  STRUCT
   S711A_B_IDLE : STRUCT
    M_AUTO_SEL : BOOL ;
    M_MANUAL_SEL : BOOL ;
    M_READY_PB : BOOL ;
    M_AUTO_RUN_PB : BOOL ;
    M_WORK_COMP_SET_PB : BOOL ;
    M_WORK_COMP_RST_PB : BOOL ;
    M_HOME_POS_PB : BOOL ;
    M_TIP_DRESS_PB : BOOL ;
    LM_SLIDE_SEL : BOOL ;
    LM_SLIDE_LOCK_SEL : BOOL ;
    LM_PIN_SEL : BOOL ;
    LM_CLAMP1_SEL : BOOL ;
    LM_CLAMP2_SEL : BOOL ;
    LM_GUN1_ADV_RET_SEL : BOOL ;
    LM_GUN2_LATCH_SEL : BOOL ;
    LM_GUN2_ADV_RET_SEL : BOOL ;
    LM_GUN1_PRESS_SEL : BOOL ;
    LM_GUN2_PRESS_SEL : BOOL ;
    LM_GUN3_PRESS_SEL : BOOL ;
    LM_IDLE_LATCH_SEL : BOOL ;
    SPARE21 : BOOL ;
    SPARE22 : BOOL ;
    SPARE23 : BOOL ;
    SPARE24 : BOOL ;
    SPARE25 : BOOL ;
    SPARE26 : BOOL ;
    SPARE27 : BOOL ;
    SPARE28 : BOOL ;
    SPARE29 : BOOL ;
    SPARE30 : BOOL ;
    M_ADV_PB : BOOL ;
    M_RET_PB : BOOL ;
    TL_SLIDE_SEL : BOOL ;
    TL_SLIDE_LOCK_SEL : BOOL ;
    TL_PIN_SEL : BOOL ;
    TL_CLAMP_SEL : BOOL ;
    TL_GUN1_ADV_RET_SEL : BOOL ;
    TL_GUN2_ADV_RET_SEL : BOOL ;
    TL_GUN3_1_ADV_RET_SEL : BOOL ;
    TL_GUN3_2_ADV_RET_SEL : BOOL ;
    TL_GUN1_PRESS_SEL : BOOL ;
    TL_GUN2_PRESS_SEL : BOOL ;
    TL_GUN3_PRESS_SEL : BOOL ;
    TL_IDLE_LATCH_SEL : BOOL ;
    SPARE46 : BOOL ;
    SPARE47 : BOOL ;
    SPARE48 : BOOL ;
    SPARE49 : BOOL ;
    SPARE50 : BOOL ;
    SPARE51 : BOOL ;
    SPARE52 : BOOL ;
    SPARE53 : BOOL ;
    SPARE54 : BOOL ;
    SPARE55 : BOOL ;
    GUN_WELD_ON : BOOL ;
    GUN_TEST_ON : BOOL ;
    LM_SELECT : BOOL ;
    TL_SELECT : BOOL ;
    SPARE60 : BOOL ;
    SPARE61 : BOOL ;
    SPARE62 : BOOL ;
    SPARE63 : BOOL ;
    SPARE64 : BOOL ;
    SPARE65 : BOOL ;
    SPARE66 : BOOL ;
    SPARE67 : BOOL ;
    SPARE68 : BOOL ;
    SPARE69 : BOOL ;
    SPARE70 : BOOL ;
    SPARE71 : BOOL ;
    SPARE72 : BOOL ;
    SPARE73 : BOOL ;
    SPARE74 : BOOL ;
    SPARE75 : BOOL ;
    SPARE76 : BOOL ;
    SPARE77 : BOOL ;
    SPARE78 : BOOL ;
    SPARE79 : BOOL ;
    SPARE80 : BOOL ;
    SPARE81 : BOOL ;
    SPARE82 : BOOL ;
    SPARE83 : BOOL ;
    SPARE84 : BOOL ;
    SPARE85 : BOOL ;
    SPARE86 : BOOL ;
    SPARE87 : BOOL ;
    SPARE88 : BOOL ;
    SPARE89 : BOOL ;
    SPARE90 : BOOL ;
    SPARE91 : BOOL ;
    SPARE92 : BOOL ;
    SPARE93 : BOOL ;
    SPARE94 : BOOL ;
    SPARE95 : BOOL ;
    SPARE96 : BOOL ;
    SPARE97 : BOOL ;
    S711A_B_LM_AS_SEL : BOOL ;
    S711A_B_TL_AS_SEL : BOOL ;
    SPARE100 : BOOL ;
    SPARE101 : BOOL ;
    SPARE102 : BOOL ;
    SPARE103 : BOOL ;
    SPARE104 : BOOL ;
    SPARE105 : BOOL ;
    SPARE106 : BOOL ;
    SPARE107 : BOOL ;
    SPARE108 : BOOL ;
    SPARE109 : BOOL ;
    SPARE110 : BOOL ;
    SPARE111 : BOOL ;
    SPARE112 : BOOL ;
    SPARE113 : BOOL ;
    SPARE114 : BOOL ;
    SPARE115 : BOOL ;
    SPARE116 : BOOL ;
    SPARE117 : BOOL ;
    SPARE118 : BOOL ;
    SPARE119 : BOOL ;
    SPARE120 : BOOL ;
    SPARE121 : BOOL ;
    SPARE122 : BOOL ;
    SPARE123 : BOOL ;
    SPARE124 : BOOL ;
    SPARE125 : BOOL ;
    SPARE126 : BOOL ;
    SPARE127 : BOOL ;
    SPARE128 : BOOL ;
    SPARE129 : BOOL ;
    SPARE130 : BOOL ;
    SPARE131 : BOOL ;
    SPARE132 : BOOL ;
    SPARE133 : BOOL ;
    SPARE134 : BOOL ;
    SPARE135 : BOOL ;
    SPARE136 : BOOL ;
    SPARE137 : BOOL ;
    SPARE138 : BOOL ;
    SPARE139 : BOOL ;
    SPARE140 : BOOL ;
    SPARE141 : BOOL ;
    SPARE142 : BOOL ;
    SPARE143 : BOOL ;
    SPARE144 : BOOL ;
    SPARE145 : BOOL ;
    SPARE146 : BOOL ;
    SPARE147 : BOOL ;
    SPARE148 : BOOL ;
    SPARE149 : BOOL ;
    SPARE150 : BOOL ;
    SPARE151 : BOOL ;
    SPARE152 : BOOL ;
    SPARE153 : BOOL ;
    SPARE154 : BOOL ;
    SPARE155 : BOOL ;
    SPARE156 : BOOL ;
    SPARE157 : BOOL ;
    SPARE158 : BOOL ;
    SPARE159 : BOOL ;
    SPARE160 : BOOL ;
    SPARE161 : BOOL ;
    LM_SLIDE_ADV_LP : WORD ;
    LM_SLIDE_RET_LP : WORD ;
    LM_SLIDE_LOCK_ADV_LP : WORD ;
    LM_SLIDE_LOCK_RET_LP : WORD ;
    LM_PIN_UP_LP : WORD ;
    LM_PIN_DOWN_LP : WORD ;
    LM_CLAMP1_ADV_LP : WORD ;
    LM_CLAMP1_RET_LP : WORD ;
    LM_CLAMP2_ADV_LP : WORD ;
    LM_CLAMP2_RET_LP : WORD ;
    LM_GUN1_ADV_LP : WORD ;
    LM_GUN1_RET_LP : WORD ;
    LM_GUN2_LATCH_ADV_LP : WORD ;
    LM_GUN2_LATCH_RET_LP : WORD ;
    LM_GUN2_ADV_LP : WORD ;
    LM_GUN2_RET_LP : WORD ;
    LM_GUN1_PRESS_LP : WORD ;
    LM_GUN1_OPEN_LP : WORD ;
    LM_GUN2_PRESS_LP : WORD ;
    LM_GUN2_OPEN_LP : WORD ;
    LM_GUN3_PRESS_LP : WORD ;
    LM_GUN3_OPEN_LP : WORD ;
    LM_IDLE_LATCH_ADV_LP : WORD ;
    LM_IDLE_LATCH_RET_LP : WORD ;
    SP_WORD36 : WORD ;
    SP_WORD37 : WORD ;
    SP_WORD38 : WORD ;
    SP_WORD39 : WORD ;
    SP_WORD40 : WORD ;
    SP_WORD41 : WORD ;
    SP_WORD42 : WORD ;
    SP_WORD43 : WORD ;
    SP_WORD44 : WORD ;
    SP_WORD45 : WORD ;
    SP_WORD46 : WORD ;
    SP_WORD47 : WORD ;
    SP_WORD48 : WORD ;
    SP_WORD49 : WORD ;
    SP_WORD50 : WORD ;
    SP_WORD51 : WORD ;
    TL_SLIDE_ADV_LP : WORD ;
    TL_SLIDE_RET_LP : WORD ;
    TL_SLIDE_LOCK_ADV_LP : WORD ;
    TL_SLIDE_LOCK_RET_LP : WORD ;
    TL_PIN_UP_LP : WORD ;
    TL_PIN_DOWN_LP : WORD ;
    TL_CLAMP1_ADV_LP : WORD ;
    TL_CLAMP1_RET_LP : WORD ;
    TL_CLAMP2_ADV_LP : WORD ;
    TL_CLAMP2_RET_LP : WORD ;
    TL_GUN1_ADV_LP : WORD ;
    TL_GUN1_RET_LP : WORD ;
    TL_GUN2_ADV_LP : WORD ;
    TL_GUN2_RET_LP : WORD ;
    TL_GUN3_1_ADV_LP : WORD ;
    TL_GUN3_1_RET_LP : WORD ;
    TL_GUN3_2_ADV_LP : WORD ;
    TL_GUN3_2_RET_LP : WORD ;
    TL_GUN1_PRESS_LP : WORD ;
    TL_GUN1_OPEN_LP : WORD ;
    TL_GUN2_PRESS_LP : WORD ;
    TL_GUN2_OPEN_LP : WORD ;
    TL_GUN3_PRESS_LP : WORD ;
    TL_GUN3_OPEN_LP : WORD ;
    TL_IDLE_PIN_UP_LP : WORD ;
    TL_IDLE_PIN_DOWN_LP : WORD ;
    TL_IDLE_LATCH_ADV_LP : WORD ;
    TL_IDLE_LATCH_RET_LP : WORD ;
    SP_WORD80 : WORD ;
    SP_WORD81 : WORD ;
    SP_WORD82 : WORD ;
    SP_WORD83 : WORD ;
    SP_WORD84 : WORD ;
    SP_WORD85 : WORD ;
    SP_WORD86 : WORD ;
    SP_WORD87 : WORD ;
    SP_WORD88 : WORD ;
    SP_WORD89 : WORD ;
    SP_WORD90 : WORD ;
    SP_WORD91 : WORD ;
    SP_WORD92 : WORD ;
    SP_WORD93 : WORD ;
    SP_WORD94 : WORD ;
    SP_WORD95 : WORD ;
    SP_WORD96 : WORD ;
    SP_WORD97 : WORD ;
    SP_WORD98 : WORD ;
    SP_WORD99 : WORD ;
    SP_WORD100 : WORD ;
    SP_WORD101 : WORD ;
   END_STRUCT ;
   S711_COMPL : STRUCT
    M_AUTO_SEL : BOOL ;
    M_MANUAL_SEL : BOOL ;
    M_READY_PB : BOOL ;
    M_AUTO_RUN_PB : BOOL ;
    M_WORK_COMP_SET_PB : BOOL ;
    M_WORK_COMP_RST_PB : BOOL ;
    M_HOME_POS_PB : BOOL ;
    M_TIP_DRESS_PB : BOOL ;
    INDEX_LOCK_SEL : BOOL ;
    INDEX_TURN_RETURN_SEL : BOOL ;
    LM_BT_CHANGE_SEL : BOOL ;
    TL_BT_CHANGE_SEL : BOOL ;
    TL_PIN_SEL : BOOL ;
    LM_PIN_SEL : BOOL ;
    LM_CLAMP_SEL : BOOL ;
    INDEX_LM_CLAMP_SEL : BOOL ;
    SPARE17 : BOOL ;
    SPARE18 : BOOL ;
    SPARE19 : BOOL ;
    SPARE20 : BOOL ;
    SPARE21 : BOOL ;
    SPARE22 : BOOL ;
    SPARE23 : BOOL ;
    SPARE24 : BOOL ;
    SPARE25 : BOOL ;
    SPARE26 : BOOL ;
    SPARE27 : BOOL ;
    SPARE28 : BOOL ;
    SPARE29 : BOOL ;
    SPARE30 : BOOL ;
    M_ADV_PB : BOOL ;
    M_RET_PB : BOOL ;
    SPARE34 : BOOL ;
    SPARE35 : BOOL ;
    SPARE36 : BOOL ;
    SPARE37 : BOOL ;
    SPARE38 : BOOL ;
    SPARE39 : BOOL ;
    SPARE40 : BOOL ;
    SPARE41 : BOOL ;
    SPARE42 : BOOL ;
    SPARE43 : BOOL ;
    SPARE44 : BOOL ;
    SPARE45 : BOOL ;
    SPARE46 : BOOL ;
    SPARE47 : BOOL ;
    SPARE48 : BOOL ;
    SPARE49 : BOOL ;
    SPARE50 : BOOL ;
    SPARE51 : BOOL ;
    SPARE52 : BOOL ;
    SPARE53 : BOOL ;
    SPARE54 : BOOL ;
    SPARE55 : BOOL ;
    SPARE56 : BOOL ;
    SPARE57 : BOOL ;
    SPARE58 : BOOL ;
    SPARE59 : BOOL ;
    SPARE60 : BOOL ;
    SPARE61 : BOOL ;
    SPARE62 : BOOL ;
    SPARE63 : BOOL ;
    SPARE64 : BOOL ;
    SPARE65 : BOOL ;
    SPARE66 : BOOL ;
    SPARE67 : BOOL ;
    SPARE68 : BOOL ;
    SPARE69 : BOOL ;
    SPARE70 : BOOL ;
    SPARE71 : BOOL ;
    SPARE72 : BOOL ;
    SPARE73 : BOOL ;
    SPARE74 : BOOL ;
    SPARE75 : BOOL ;
    SPARE76 : BOOL ;
    SPARE77 : BOOL ;
    SPARE78 : BOOL ;
    SPARE79 : BOOL ;
    SPARE80 : BOOL ;
    SPARE81 : BOOL ;
    SPARE82 : BOOL ;
    SPARE83 : BOOL ;
    SPARE84 : BOOL ;
    SPARE85 : BOOL ;
    SPARE86 : BOOL ;
    SPARE87 : BOOL ;
    SPARE88 : BOOL ;
    SPARE89 : BOOL ;
    SPARE90 : BOOL ;
    SPARE91 : BOOL ;
    SPARE92 : BOOL ;
    SPARE93 : BOOL ;
    SPARE94 : BOOL ;
    SPARE95 : BOOL ;
    SPARE96 : BOOL ;
    SPARE97 : BOOL ;
    SPARE98 : BOOL ;
    SPARE99 : BOOL ;
    SPARE100 : BOOL ;
    SPARE101 : BOOL ;
    SPARE102 : BOOL ;
    SPARE103 : BOOL ;
    SPARE104 : BOOL ;
    SPARE105 : BOOL ;
    SPARE106 : BOOL ;
    SPARE107 : BOOL ;
    SPARE108 : BOOL ;
    SPARE109 : BOOL ;
    SPARE110 : BOOL ;
    SPARE111 : BOOL ;
    SPARE112 : BOOL ;
    SPARE113 : BOOL ;
    SPARE114 : BOOL ;
    SPARE115 : BOOL ;
    SPARE116 : BOOL ;
    SPARE117 : BOOL ;
    SPARE118 : BOOL ;
    SPARE119 : BOOL ;
    SPARE120 : BOOL ;
    SPARE121 : BOOL ;
    SPARE122 : BOOL ;
    SPARE123 : BOOL ;
    SPARE124 : BOOL ;
    SPARE125 : BOOL ;
    SPARE126 : BOOL ;
    SPARE127 : BOOL ;
    SPARE128 : BOOL ;
    SPARE129 : BOOL ;
    SPARE130 : BOOL ;
    SPARE131 : BOOL ;
    SPARE132 : BOOL ;
    SPARE133 : BOOL ;
    SPARE134 : BOOL ;
    SPARE135 : BOOL ;
    SPARE136 : BOOL ;
    SPARE137 : BOOL ;
    SPARE138 : BOOL ;
    SPARE139 : BOOL ;
    SPARE140 : BOOL ;
    SPARE141 : BOOL ;
    SPARE142 : BOOL ;
    SPARE143 : BOOL ;
    SPARE144 : BOOL ;
    SPARE145 : BOOL ;
    SPARE146 : BOOL ;
    SPARE147 : BOOL ;
    SPARE148 : BOOL ;
    SPARE149 : BOOL ;
    SPARE150 : BOOL ;
    SPARE151 : BOOL ;
    SPARE152 : BOOL ;
    SPARE153 : BOOL ;
    SPARE154 : BOOL ;
    SPARE155 : BOOL ;
    SPARE156 : BOOL ;
    SPARE157 : BOOL ;
    SPARE158 : BOOL ;
    SPARE159 : BOOL ;
    SPARE160 : BOOL ;
    SPARE161 : BOOL ;
    INDEX_LOCK_ADV_LP : WORD ;
    INDEX_LOCK_RET_LP : WORD ;
    INDEX_TURN_LP : WORD ;
    INDEX_RETURN_LP : WORD ;
    LM_BT_CHANGE_ADV_LP : WORD ;
    LM_BT_CHANGE_RET_LP : WORD ;
    TL_BT_CHANGE_ADV_LP : WORD ;
    TL_BT_CHANGE_RET_LP : WORD ;
    TL_PIN_UP_LP : WORD ;
    TL_PIN_DOWN_LP : WORD ;
    LM_PIN_UP_LP : WORD ;
    LM_PIN_DOWN_LP : WORD ;
    LM_CLAMP_ADV_LP : WORD ;
    LM_CLAMP_RET_LP : WORD ;
    INDEX_LM_CLAMP_ADV_LP : WORD ;
    INDEX_LM_CLAMP_RET_LP : WORD ;
    INDEX_LM_PIN_UP_LP : WORD ;
    INDEX_LM_PIN_DOWN_LP : WORD ;
    SP_WORD29 : WORD ;
    SP_WORD30 : WORD ;
    SP_WORD31 : WORD ;
    SP_WORD32 : WORD ;
    SP_WORD33 : WORD ;
    SP_WORD34 : WORD ;
    SP_WORD35 : WORD ;
    SP_WORD36 : WORD ;
    SP_WORD37 : WORD ;
    SP_WORD38 : WORD ;
    SP_WORD39 : WORD ;
    SP_WORD40 : WORD ;
    SP_WORD41 : WORD ;
    SP_WORD42 : WORD ;
    SP_WORD43 : WORD ;
    SP_WORD44 : WORD ;
    SP_WORD45 : WORD ;
    SP_WORD46 : WORD ;
    SP_WORD47 : WORD ;
    SP_WORD49 : WORD ;
    SP_WORD50 : WORD ;
    SP_WORD51 : WORD ;
    INR_PLT3_UP_LP : WORD ;
    INR_PLT3_DOWN_LP : WORD ;
    INR_PLT3_LOCK_ADV_LP : WORD ;
    INR_PLT3_LOCK_RET_LP : WORD ;
    INR_PLT4_UP_LP : WORD ;
    INR_PLT4_DOWN_LP : WORD ;
    INR_PLT4_LOCK_ADV_LP : WORD ;
    INR_PLT4_LOCK_RET_LP : WORD ;
    INR_PLT5_UP_LP : WORD ;
    INR_PLT5_DOWN_LP : WORD ;
    INR_PLT5_LOCK_ADV_LP : WORD ;
    INR_PLT5_LOCK_RET_LP : WORD ;
    SP_WORD64 : WORD ;
    SP_WORD65 : WORD ;
    SP_WORD66 : WORD ;
    SP_WORD67 : WORD ;
    SP_WORD68 : WORD ;
    SP_WORD69 : WORD ;
    SP_WORD70 : WORD ;
    SP_WORD71 : WORD ;
    SP_WORD72 : WORD ;
    SP_WORD73 : WORD ;
    SP_WORD74 : WORD ;
    SP_WORD75 : WORD ;
    SP_WORD76 : WORD ;
    SP_WORD77 : WORD ;
    SP_WORD78 : WORD ;
    SP_WORD79 : WORD ;
    SP_WORD80 : WORD ;
    SP_WORD81 : WORD ;
    SP_WORD82 : WORD ;
    SP_WORD83 : WORD ;
    SP_WORD84 : WORD ;
    SP_WORD85 : WORD ;
    SP_WORD86 : WORD ;
    SP_WORD87 : WORD ;
    SP_WORD88 : WORD ;
    SP_WORD89 : WORD ;
    SP_WORD90 : WORD ;
    SP_WORD91 : WORD ;
    SP_WORD92 : WORD ;
    SP_WORD93 : WORD ;
    SP_WORD94 : WORD ;
    SP_WORD95 : WORD ;
    SP_WORD96 : WORD ;
    SP_WORD97 : WORD ;
    SP_WORD98 : WORD ;
    SP_WORD99 : WORD ;
    SP_WORD100 : WORD ;
    SP_WORD101 : WORD ;
   END_STRUCT ;
  END_STRUCT ;
BEGIN
   S711A_B_IDLE.M_AUTO_SEL := FALSE;
   S711A_B_IDLE.M_MANUAL_SEL := FALSE;
   S711A_B_IDLE.M_READY_PB := FALSE;
   S711A_B_IDLE.M_AUTO_RUN_PB := FALSE;
   S711A_B_IDLE.M_WORK_COMP_SET_PB := FALSE;
   S711A_B_IDLE.M_WORK_COMP_RST_PB := FALSE;
   S711A_B_IDLE.M_HOME_POS_PB := FALSE;
   S711A_B_IDLE.M_TIP_DRESS_PB := FALSE;
   S711A_B_IDLE.LM_SLIDE_SEL := FALSE;
   S711A_B_IDLE.LM_SLIDE_LOCK_SEL := FALSE;
   S711A_B_IDLE.LM_PIN_SEL := FALSE;
   S711A_B_IDLE.LM_CLAMP1_SEL := FALSE;
   S711A_B_IDLE.LM_CLAMP2_SEL := FALSE;
   S711A_B_IDLE.LM_GUN1_ADV_RET_SEL := FALSE;
   S711A_B_IDLE.LM_GUN2_LATCH_SEL := FALSE;
   S711A_B_IDLE.LM_GUN2_ADV_RET_SEL := FALSE;
   S711A_B_IDLE.LM_GUN1_PRESS_SEL := FALSE;
   S711A_B_IDLE.LM_GUN2_PRESS_SEL := FALSE;
   S711A_B_IDLE.LM_GUN3_PRESS_SEL := FALSE;
   S711A_B_IDLE.LM_IDLE_LATCH_SEL := FALSE;
   S711A_B_IDLE.SPARE21 := FALSE;
   S711A_B_IDLE.SPARE22 := FALSE;
   S711A_B_IDLE.SPARE23 := FALSE;
   S711A_B_IDLE.SPARE24 := FALSE;
   S711A_B_IDLE.SPARE25 := FALSE;
   S711A_B_IDLE.SPARE26 := FALSE;
   S711A_B_IDLE.SPARE27 := FALSE;
   S711A_B_IDLE.SPARE28 := FALSE;
   S711A_B_IDLE.SPARE29 := FALSE;
   S711A_B_IDLE.SPARE30 := FALSE;
   S711A_B_IDLE.M_ADV_PB := FALSE;
   S711A_B_IDLE.M_RET_PB := FALSE;
   S711A_B_IDLE.TL_SLIDE_SEL := FALSE;
   S711A_B_IDLE.TL_SLIDE_LOCK_SEL := FALSE;
   S711A_B_IDLE.TL_PIN_SEL := FALSE;
   S711A_B_IDLE.TL_CLAMP_SEL := FALSE;
   S711A_B_IDLE.TL_GUN1_ADV_RET_SEL := FALSE;
   S711A_B_IDLE.TL_GUN2_ADV_RET_SEL := FALSE;
   S711A_B_IDLE.TL_GUN3_1_ADV_RET_SEL := FALSE;
   S711A_B_IDLE.TL_GUN3_2_ADV_RET_SEL := FALSE;
   S711A_B_IDLE.TL_GUN1_PRESS_SEL := FALSE;
   S711A_B_IDLE.TL_GUN2_PRESS_SEL := FALSE;
   S711A_B_IDLE.TL_GUN3_PRESS_SEL := FALSE;
   S711A_B_IDLE.TL_IDLE_LATCH_SEL := FALSE;
   S711A_B_IDLE.SPARE46 := FALSE;
   S711A_B_IDLE.SPARE47 := FALSE;
   S711A_B_IDLE.SPARE48 := FALSE;
   S711A_B_IDLE.SPARE49 := FALSE;
   S711A_B_IDLE.SPARE50 := FALSE;
   S711A_B_IDLE.SPARE51 := FALSE;
   S711A_B_IDLE.SPARE52 := FALSE;
   S711A_B_IDLE.SPARE53 := FALSE;
   S711A_B_IDLE.SPARE54 := FALSE;
   S711A_B_IDLE.SPARE55 := FALSE;
   S711A_B_IDLE.GUN_WELD_ON := FALSE;
   S711A_B_IDLE.GUN_TEST_ON := FALSE;
   S711A_B_IDLE.LM_SELECT := FALSE;
   S711A_B_IDLE.TL_SELECT := FALSE;
   S711A_B_IDLE.SPARE60 := FALSE;
   S711A_B_IDLE.SPARE61 := FALSE;
   S711A_B_IDLE.SPARE62 := FALSE;
   S711A_B_IDLE.SPARE63 := FALSE;
   S711A_B_IDLE.SPARE64 := FALSE;
   S711A_B_IDLE.SPARE65 := FALSE;
   S711A_B_IDLE.SPARE66 := FALSE;
   S711A_B_IDLE.SPARE67 := FALSE;
   S711A_B_IDLE.SPARE68 := FALSE;
   S711A_B_IDLE.SPARE69 := FALSE;
   S711A_B_IDLE.SPARE70 := FALSE;
   S711A_B_IDLE.SPARE71 := FALSE;
   S711A_B_IDLE.SPARE72 := FALSE;
   S711A_B_IDLE.SPARE73 := FALSE;
   S711A_B_IDLE.SPARE74 := FALSE;
   S711A_B_IDLE.SPARE75 := FALSE;
   S711A_B_IDLE.SPARE76 := FALSE;
   S711A_B_IDLE.SPARE77 := FALSE;
   S711A_B_IDLE.SPARE78 := FALSE;
   S711A_B_IDLE.SPARE79 := FALSE;
   S711A_B_IDLE.SPARE80 := FALSE;
   S711A_B_IDLE.SPARE81 := FALSE;
   S711A_B_IDLE.SPARE82 := FALSE;
   S711A_B_IDLE.SPARE83 := FALSE;
   S711A_B_IDLE.SPARE84 := FALSE;
   S711A_B_IDLE.SPARE85 := FALSE;
   S711A_B_IDLE.SPARE86 := FALSE;
   S711A_B_IDLE.SPARE87 := FALSE;
   S711A_B_IDLE.SPARE88 := FALSE;
   S711A_B_IDLE.SPARE89 := FALSE;
   S711A_B_IDLE.SPARE90 := FALSE;
   S711A_B_IDLE.SPARE91 := FALSE;
   S711A_B_IDLE.SPARE92 := FALSE;
   S711A_B_IDLE.SPARE93 := FALSE;
   S711A_B_IDLE.SPARE94 := FALSE;
   S711A_B_IDLE.SPARE95 := FALSE;
   S711A_B_IDLE.SPARE96 := FALSE;
   S711A_B_IDLE.SPARE97 := FALSE;
   S711A_B_IDLE.S711A_B_LM_AS_SEL := FALSE;
   S711A_B_IDLE.S711A_B_TL_AS_SEL := FALSE;
   S711A_B_IDLE.SPARE100 := FALSE;
   S711A_B_IDLE.SPARE101 := FALSE;
   S711A_B_IDLE.SPARE102 := FALSE;
   S711A_B_IDLE.SPARE103 := FALSE;
   S711A_B_IDLE.SPARE104 := FALSE;
   S711A_B_IDLE.SPARE105 := FALSE;
   S711A_B_IDLE.SPARE106 := FALSE;
   S711A_B_IDLE.SPARE107 := FALSE;
   S711A_B_IDLE.SPARE108 := FALSE;
   S711A_B_IDLE.SPARE109 := FALSE;
   S711A_B_IDLE.SPARE110 := FALSE;
   S711A_B_IDLE.SPARE111 := FALSE;
   S711A_B_IDLE.SPARE112 := FALSE;
   S711A_B_IDLE.SPARE113 := FALSE;
   S711A_B_IDLE.SPARE114 := FALSE;
   S711A_B_IDLE.SPARE115 := FALSE;
   S711A_B_IDLE.SPARE116 := FALSE;
   S711A_B_IDLE.SPARE117 := FALSE;
   S711A_B_IDLE.SPARE118 := FALSE;
   S711A_B_IDLE.SPARE119 := FALSE;
   S711A_B_IDLE.SPARE120 := FALSE;
   S711A_B_IDLE.SPARE121 := FALSE;
   S711A_B_IDLE.SPARE122 := FALSE;
   S711A_B_IDLE.SPARE123 := FALSE;
   S711A_B_IDLE.SPARE124 := FALSE;
   S711A_B_IDLE.SPARE125 := FALSE;
   S711A_B_IDLE.SPARE126 := FALSE;
   S711A_B_IDLE.SPARE127 := FALSE;
   S711A_B_IDLE.SPARE128 := FALSE;
   S711A_B_IDLE.SPARE129 := FALSE;
   S711A_B_IDLE.SPARE130 := FALSE;
   S711A_B_IDLE.SPARE131 := FALSE;
   S711A_B_IDLE.SPARE132 := FALSE;
   S711A_B_IDLE.SPARE133 := FALSE;
   S711A_B_IDLE.SPARE134 := FALSE;
   S711A_B_IDLE.SPARE135 := FALSE;
   S711A_B_IDLE.SPARE136 := FALSE;
   S711A_B_IDLE.SPARE137 := FALSE;
   S711A_B_IDLE.SPARE138 := FALSE;
   S711A_B_IDLE.SPARE139 := FALSE;
   S711A_B_IDLE.SPARE140 := FALSE;
   S711A_B_IDLE.SPARE141 := FALSE;
   S711A_B_IDLE.SPARE142 := FALSE;
   S711A_B_IDLE.SPARE143 := FALSE;
   S711A_B_IDLE.SPARE144 := FALSE;
   S711A_B_IDLE.SPARE145 := FALSE;
   S711A_B_IDLE.SPARE146 := FALSE;
   S711A_B_IDLE.SPARE147 := FALSE;
   S711A_B_IDLE.SPARE148 := FALSE;
   S711A_B_IDLE.SPARE149 := FALSE;
   S711A_B_IDLE.SPARE150 := FALSE;
   S711A_B_IDLE.SPARE151 := FALSE;
   S711A_B_IDLE.SPARE152 := FALSE;
   S711A_B_IDLE.SPARE153 := FALSE;
   S711A_B_IDLE.SPARE154 := FALSE;
   S711A_B_IDLE.SPARE155 := FALSE;
   S711A_B_IDLE.SPARE156 := FALSE;
   S711A_B_IDLE.SPARE157 := FALSE;
   S711A_B_IDLE.SPARE158 := FALSE;
   S711A_B_IDLE.SPARE159 := FALSE;
   S711A_B_IDLE.SPARE160 := FALSE;
   S711A_B_IDLE.SPARE161 := FALSE;
   S711A_B_IDLE.LM_SLIDE_ADV_LP := W#16#0;
   S711A_B_IDLE.LM_SLIDE_RET_LP := W#16#0;
   S711A_B_IDLE.LM_SLIDE_LOCK_ADV_LP := W#16#0;
   S711A_B_IDLE.LM_SLIDE_LOCK_RET_LP := W#16#0;
   S711A_B_IDLE.LM_PIN_UP_LP := W#16#0;
   S711A_B_IDLE.LM_PIN_DOWN_LP := W#16#0;
   S711A_B_IDLE.LM_CLAMP1_ADV_LP := W#16#0;
   S711A_B_IDLE.LM_CLAMP1_RET_LP := W#16#0;
   S711A_B_IDLE.LM_CLAMP2_ADV_LP := W#16#0;
   S711A_B_IDLE.LM_CLAMP2_RET_LP := W#16#0;
   S711A_B_IDLE.LM_GUN1_ADV_LP := W#16#0;
   S711A_B_IDLE.LM_GUN1_RET_LP := W#16#0;
   S711A_B_IDLE.LM_GUN2_LATCH_ADV_LP := W#16#0;
   S711A_B_IDLE.LM_GUN2_LATCH_RET_LP := W#16#0;
   S711A_B_IDLE.LM_GUN2_ADV_LP := W#16#0;
   S711A_B_IDLE.LM_GUN2_RET_LP := W#16#0;
   S711A_B_IDLE.LM_GUN1_PRESS_LP := W#16#0;
   S711A_B_IDLE.LM_GUN1_OPEN_LP := W#16#0;
   S711A_B_IDLE.LM_GUN2_PRESS_LP := W#16#0;
   S711A_B_IDLE.LM_GUN2_OPEN_LP := W#16#0;
   S711A_B_IDLE.LM_GUN3_PRESS_LP := W#16#0;
   S711A_B_IDLE.LM_GUN3_OPEN_LP := W#16#0;
   S711A_B_IDLE.LM_IDLE_LATCH_ADV_LP := W#16#0;
   S711A_B_IDLE.LM_IDLE_LATCH_RET_LP := W#16#0;
   S711A_B_IDLE.SP_WORD36 := W#16#0;
   S711A_B_IDLE.SP_WORD37 := W#16#0;
   S711A_B_IDLE.SP_WORD38 := W#16#0;
   S711A_B_IDLE.SP_WORD39 := W#16#0;
   S711A_B_IDLE.SP_WORD40 := W#16#0;
   S711A_B_IDLE.SP_WORD41 := W#16#0;
   S711A_B_IDLE.SP_WORD42 := W#16#0;
   S711A_B_IDLE.SP_WORD43 := W#16#0;
   S711A_B_IDLE.SP_WORD44 := W#16#0;
   S711A_B_IDLE.SP_WORD45 := W#16#0;
   S711A_B_IDLE.SP_WORD46 := W#16#0;
   S711A_B_IDLE.SP_WORD47 := W#16#0;
   S711A_B_IDLE.SP_WORD48 := W#16#0;
   S711A_B_IDLE.SP_WORD49 := W#16#0;
   S711A_B_IDLE.SP_WORD50 := W#16#0;
   S711A_B_IDLE.SP_WORD51 := W#16#0;
   S711A_B_IDLE.TL_SLIDE_ADV_LP := W#16#0;
   S711A_B_IDLE.TL_SLIDE_RET_LP := W#16#0;
   S711A_B_IDLE.TL_SLIDE_LOCK_ADV_LP := W#16#0;
   S711A_B_IDLE.TL_SLIDE_LOCK_RET_LP := W#16#0;
   S711A_B_IDLE.TL_PIN_UP_LP := W#16#0;
   S711A_B_IDLE.TL_PIN_DOWN_LP := W#16#0;
   S711A_B_IDLE.TL_CLAMP1_ADV_LP := W#16#0;
   S711A_B_IDLE.TL_CLAMP1_RET_LP := W#16#0;
   S711A_B_IDLE.TL_CLAMP2_ADV_LP := W#16#0;
   S711A_B_IDLE.TL_CLAMP2_RET_LP := W#16#0;
   S711A_B_IDLE.TL_GUN1_ADV_LP := W#16#0;
   S711A_B_IDLE.TL_GUN1_RET_LP := W#16#0;
   S711A_B_IDLE.TL_GUN2_ADV_LP := W#16#0;
   S711A_B_IDLE.TL_GUN2_RET_LP := W#16#0;
   S711A_B_IDLE.TL_GUN3_1_ADV_LP := W#16#0;
   S711A_B_IDLE.TL_GUN3_1_RET_LP := W#16#0;
   S711A_B_IDLE.TL_GUN3_2_ADV_LP := W#16#0;
   S711A_B_IDLE.TL_GUN3_2_RET_LP := W#16#0;
   S711A_B_IDLE.TL_GUN1_PRESS_LP := W#16#0;
   S711A_B_IDLE.TL_GUN1_OPEN_LP := W#16#0;
   S711A_B_IDLE.TL_GUN2_PRESS_LP := W#16#0;
   S711A_B_IDLE.TL_GUN2_OPEN_LP := W#16#0;
   S711A_B_IDLE.TL_GUN3_PRESS_LP := W#16#0;
   S711A_B_IDLE.TL_GUN3_OPEN_LP := W#16#0;
   S711A_B_IDLE.TL_IDLE_PIN_UP_LP := W#16#0;
   S711A_B_IDLE.TL_IDLE_PIN_DOWN_LP := W#16#0;
   S711A_B_IDLE.TL_IDLE_LATCH_ADV_LP := W#16#0;
   S711A_B_IDLE.TL_IDLE_LATCH_RET_LP := W#16#0;
   S711A_B_IDLE.SP_WORD80 := W#16#0;
   S711A_B_IDLE.SP_WORD81 := W#16#0;
   S711A_B_IDLE.SP_WORD82 := W#16#0;
   S711A_B_IDLE.SP_WORD83 := W#16#0;
   S711A_B_IDLE.SP_WORD84 := W#16#0;
   S711A_B_IDLE.SP_WORD85 := W#16#0;
   S711A_B_IDLE.SP_WORD86 := W#16#0;
   S711A_B_IDLE.SP_WORD87 := W#16#0;
   S711A_B_IDLE.SP_WORD88 := W#16#0;
   S711A_B_IDLE.SP_WORD89 := W#16#0;
   S711A_B_IDLE.SP_WORD90 := W#16#0;
   S711A_B_IDLE.SP_WORD91 := W#16#0;
   S711A_B_IDLE.SP_WORD92 := W#16#0;
   S711A_B_IDLE.SP_WORD93 := W#16#0;
   S711A_B_IDLE.SP_WORD94 := W#16#0;
   S711A_B_IDLE.SP_WORD95 := W#16#0;
   S711A_B_IDLE.SP_WORD96 := W#16#0;
   S711A_B_IDLE.SP_WORD97 := W#16#0;
   S711A_B_IDLE.SP_WORD98 := W#16#0;
   S711A_B_IDLE.SP_WORD99 := W#16#0;
   S711A_B_IDLE.SP_WORD100 := W#16#0;
   S711A_B_IDLE.SP_WORD101 := W#16#0;
   S711_COMPL.M_AUTO_SEL := FALSE;
   S711_COMPL.M_MANUAL_SEL := FALSE;
   S711_COMPL.M_READY_PB := FALSE;
   S711_COMPL.M_AUTO_RUN_PB := FALSE;
   S711_COMPL.M_WORK_COMP_SET_PB := FALSE;
   S711_COMPL.M_WORK_COMP_RST_PB := FALSE;
   S711_COMPL.M_HOME_POS_PB := FALSE;
   S711_COMPL.M_TIP_DRESS_PB := FALSE;
   S711_COMPL.INDEX_LOCK_SEL := FALSE;
   S711_COMPL.INDEX_TURN_RETURN_SEL := FALSE;
   S711_COMPL.LM_BT_CHANGE_SEL := FALSE;
   S711_COMPL.TL_BT_CHANGE_SEL := FALSE;
   S711_COMPL.TL_PIN_SEL := FALSE;
   S711_COMPL.LM_PIN_SEL := FALSE;
   S711_COMPL.LM_CLAMP_SEL := FALSE;
   S711_COMPL.INDEX_LM_CLAMP_SEL := FALSE;
   S711_COMPL.SPARE17 := FALSE;
   S711_COMPL.SPARE18 := FALSE;
   S711_COMPL.SPARE19 := FALSE;
   S711_COMPL.SPARE20 := FALSE;
   S711_COMPL.SPARE21 := FALSE;
   S711_COMPL.SPARE22 := FALSE;
   S711_COMPL.SPARE23 := FALSE;
   S711_COMPL.SPARE24 := FALSE;
   S711_COMPL.SPARE25 := FALSE;
   S711_COMPL.SPARE26 := FALSE;
   S711_COMPL.SPARE27 := FALSE;
   S711_COMPL.SPARE28 := FALSE;
   S711_COMPL.SPARE29 := FALSE;
   S711_COMPL.SPARE30 := FALSE;
   S711_COMPL.M_ADV_PB := FALSE;
   S711_COMPL.M_RET_PB := FALSE;
   S711_COMPL.SPARE34 := FALSE;
   S711_COMPL.SPARE35 := FALSE;
   S711_COMPL.SPARE36 := FALSE;
   S711_COMPL.SPARE37 := FALSE;
   S711_COMPL.SPARE38 := FALSE;
   S711_COMPL.SPARE39 := FALSE;
   S711_COMPL.SPARE40 := FALSE;
   S711_COMPL.SPARE41 := FALSE;
   S711_COMPL.SPARE42 := FALSE;
   S711_COMPL.SPARE43 := FALSE;
   S711_COMPL.SPARE44 := FALSE;
   S711_COMPL.SPARE45 := FALSE;
   S711_COMPL.SPARE46 := FALSE;
   S711_COMPL.SPARE47 := FALSE;
   S711_COMPL.SPARE48 := FALSE;
   S711_COMPL.SPARE49 := FALSE;
   S711_COMPL.SPARE50 := FALSE;
   S711_COMPL.SPARE51 := FALSE;
   S711_COMPL.SPARE52 := FALSE;
   S711_COMPL.SPARE53 := FALSE;
   S711_COMPL.SPARE54 := FALSE;
   S711_COMPL.SPARE55 := FALSE;
   S711_COMPL.SPARE56 := FALSE;
   S711_COMPL.SPARE57 := FALSE;
   S711_COMPL.SPARE58 := FALSE;
   S711_COMPL.SPARE59 := FALSE;
   S711_COMPL.SPARE60 := FALSE;
   S711_COMPL.SPARE61 := FALSE;
   S711_COMPL.SPARE62 := FALSE;
   S711_COMPL.SPARE63 := FALSE;
   S711_COMPL.SPARE64 := FALSE;
   S711_COMPL.SPARE65 := FALSE;
   S711_COMPL.SPARE66 := FALSE;
   S711_COMPL.SPARE67 := FALSE;
   S711_COMPL.SPARE68 := FALSE;
   S711_COMPL.SPARE69 := FALSE;
   S711_COMPL.SPARE70 := FALSE;
   S711_COMPL.SPARE71 := FALSE;
   S711_COMPL.SPARE72 := FALSE;
   S711_COMPL.SPARE73 := FALSE;
   S711_COMPL.SPARE74 := FALSE;
   S711_COMPL.SPARE75 := FALSE;
   S711_COMPL.SPARE76 := FALSE;
   S711_COMPL.SPARE77 := FALSE;
   S711_COMPL.SPARE78 := FALSE;
   S711_COMPL.SPARE79 := FALSE;
   S711_COMPL.SPARE80 := FALSE;
   S711_COMPL.SPARE81 := FALSE;
   S711_COMPL.SPARE82 := FALSE;
   S711_COMPL.SPARE83 := FALSE;
   S711_COMPL.SPARE84 := FALSE;
   S711_COMPL.SPARE85 := FALSE;
   S711_COMPL.SPARE86 := FALSE;
   S711_COMPL.SPARE87 := FALSE;
   S711_COMPL.SPARE88 := FALSE;
   S711_COMPL.SPARE89 := FALSE;
   S711_COMPL.SPARE90 := FALSE;
   S711_COMPL.SPARE91 := FALSE;
   S711_COMPL.SPARE92 := FALSE;
   S711_COMPL.SPARE93 := FALSE;
   S711_COMPL.SPARE94 := FALSE;
   S711_COMPL.SPARE95 := FALSE;
   S711_COMPL.SPARE96 := FALSE;
   S711_COMPL.SPARE97 := FALSE;
   S711_COMPL.SPARE98 := FALSE;
   S711_COMPL.SPARE99 := FALSE;
   S711_COMPL.SPARE100 := FALSE;
   S711_COMPL.SPARE101 := FALSE;
   S711_COMPL.SPARE102 := FALSE;
   S711_COMPL.SPARE103 := FALSE;
   S711_COMPL.SPARE104 := FALSE;
   S711_COMPL.SPARE105 := FALSE;
   S711_COMPL.SPARE106 := FALSE;
   S711_COMPL.SPARE107 := FALSE;
   S711_COMPL.SPARE108 := FALSE;
   S711_COMPL.SPARE109 := FALSE;
   S711_COMPL.SPARE110 := FALSE;
   S711_COMPL.SPARE111 := FALSE;
   S711_COMPL.SPARE112 := FALSE;
   S711_COMPL.SPARE113 := FALSE;
   S711_COMPL.SPARE114 := FALSE;
   S711_COMPL.SPARE115 := FALSE;
   S711_COMPL.SPARE116 := FALSE;
   S711_COMPL.SPARE117 := FALSE;
   S711_COMPL.SPARE118 := FALSE;
   S711_COMPL.SPARE119 := FALSE;
   S711_COMPL.SPARE120 := FALSE;
   S711_COMPL.SPARE121 := FALSE;
   S711_COMPL.SPARE122 := FALSE;
   S711_COMPL.SPARE123 := FALSE;
   S711_COMPL.SPARE124 := FALSE;
   S711_COMPL.SPARE125 := FALSE;
   S711_COMPL.SPARE126 := FALSE;
   S711_COMPL.SPARE127 := FALSE;
   S711_COMPL.SPARE128 := FALSE;
   S711_COMPL.SPARE129 := FALSE;
   S711_COMPL.SPARE130 := FALSE;
   S711_COMPL.SPARE131 := FALSE;
   S711_COMPL.SPARE132 := FALSE;
   S711_COMPL.SPARE133 := FALSE;
   S711_COMPL.SPARE134 := FALSE;
   S711_COMPL.SPARE135 := FALSE;
   S711_COMPL.SPARE136 := FALSE;
   S711_COMPL.SPARE137 := FALSE;
   S711_COMPL.SPARE138 := FALSE;
   S711_COMPL.SPARE139 := FALSE;
   S711_COMPL.SPARE140 := FALSE;
   S711_COMPL.SPARE141 := FALSE;
   S711_COMPL.SPARE142 := FALSE;
   S711_COMPL.SPARE143 := FALSE;
   S711_COMPL.SPARE144 := FALSE;
   S711_COMPL.SPARE145 := FALSE;
   S711_COMPL.SPARE146 := FALSE;
   S711_COMPL.SPARE147 := FALSE;
   S711_COMPL.SPARE148 := FALSE;
   S711_COMPL.SPARE149 := FALSE;
   S711_COMPL.SPARE150 := FALSE;
   S711_COMPL.SPARE151 := FALSE;
   S711_COMPL.SPARE152 := FALSE;
   S711_COMPL.SPARE153 := FALSE;
   S711_COMPL.SPARE154 := FALSE;
   S711_COMPL.SPARE155 := FALSE;
   S711_COMPL.SPARE156 := FALSE;
   S711_COMPL.SPARE157 := FALSE;
   S711_COMPL.SPARE158 := FALSE;
   S711_COMPL.SPARE159 := FALSE;
   S711_COMPL.SPARE160 := FALSE;
   S711_COMPL.SPARE161 := FALSE;
   S711_COMPL.INDEX_LOCK_ADV_LP := W#16#0;
   S711_COMPL.INDEX_LOCK_RET_LP := W#16#0;
   S711_COMPL.INDEX_TURN_LP := W#16#0;
   S711_COMPL.INDEX_RETURN_LP := W#16#0;
   S711_COMPL.LM_BT_CHANGE_ADV_LP := W#16#0;
   S711_COMPL.LM_BT_CHANGE_RET_LP := W#16#0;
   S711_COMPL.TL_BT_CHANGE_ADV_LP := W#16#0;
   S711_COMPL.TL_BT_CHANGE_RET_LP := W#16#0;
   S711_COMPL.TL_PIN_UP_LP := W#16#0;
   S711_COMPL.TL_PIN_DOWN_LP := W#16#0;
   S711_COMPL.LM_PIN_UP_LP := W#16#0;
   S711_COMPL.LM_PIN_DOWN_LP := W#16#0;
   S711_COMPL.LM_CLAMP_ADV_LP := W#16#0;
   S711_COMPL.LM_CLAMP_RET_LP := W#16#0;
   S711_COMPL.INDEX_LM_CLAMP_ADV_LP := W#16#0;
   S711_COMPL.INDEX_LM_CLAMP_RET_LP := W#16#0;
   S711_COMPL.INDEX_LM_PIN_UP_LP := W#16#0;
   S711_COMPL.INDEX_LM_PIN_DOWN_LP := W#16#0;
   S711_COMPL.SP_WORD29 := W#16#0;
   S711_COMPL.SP_WORD30 := W#16#0;
   S711_COMPL.SP_WORD31 := W#16#0;
   S711_COMPL.SP_WORD32 := W#16#0;
   S711_COMPL.SP_WORD33 := W#16#0;
   S711_COMPL.SP_WORD34 := W#16#0;
   S711_COMPL.SP_WORD35 := W#16#0;
   S711_COMPL.SP_WORD36 := W#16#0;
   S711_COMPL.SP_WORD37 := W#16#0;
   S711_COMPL.SP_WORD38 := W#16#0;
   S711_COMPL.SP_WORD39 := W#16#0;
   S711_COMPL.SP_WORD40 := W#16#0;
   S711_COMPL.SP_WORD41 := W#16#0;
   S711_COMPL.SP_WORD42 := W#16#0;
   S711_COMPL.SP_WORD43 := W#16#0;
   S711_COMPL.SP_WORD44 := W#16#0;
   S711_COMPL.SP_WORD45 := W#16#0;
   S711_COMPL.SP_WORD46 := W#16#0;
   S711_COMPL.SP_WORD47 := W#16#0;
   S711_COMPL.SP_WORD49 := W#16#0;
   S711_COMPL.SP_WORD50 := W#16#0;
   S711_COMPL.SP_WORD51 := W#16#0;
   S711_COMPL.INR_PLT3_UP_LP := W#16#0;
   S711_COMPL.INR_PLT3_DOWN_LP := W#16#0;
   S711_COMPL.INR_PLT3_LOCK_ADV_LP := W#16#0;
   S711_COMPL.INR_PLT3_LOCK_RET_LP := W#16#0;
   S711_COMPL.INR_PLT4_UP_LP := W#16#0;
   S711_COMPL.INR_PLT4_DOWN_LP := W#16#0;
   S711_COMPL.INR_PLT4_LOCK_ADV_LP := W#16#0;
   S711_COMPL.INR_PLT4_LOCK_RET_LP := W#16#0;
   S711_COMPL.INR_PLT5_UP_LP := W#16#0;
   S711_COMPL.INR_PLT5_DOWN_LP := W#16#0;
   S711_COMPL.INR_PLT5_LOCK_ADV_LP := W#16#0;
   S711_COMPL.INR_PLT5_LOCK_RET_LP := W#16#0;
   S711_COMPL.SP_WORD64 := W#16#0;
   S711_COMPL.SP_WORD65 := W#16#0;
   S711_COMPL.SP_WORD66 := W#16#0;
   S711_COMPL.SP_WORD67 := W#16#0;
   S711_COMPL.SP_WORD68 := W#16#0;
   S711_COMPL.SP_WORD69 := W#16#0;
   S711_COMPL.SP_WORD70 := W#16#0;
   S711_COMPL.SP_WORD71 := W#16#0;
   S711_COMPL.SP_WORD72 := W#16#0;
   S711_COMPL.SP_WORD73 := W#16#0;
   S711_COMPL.SP_WORD74 := W#16#0;
   S711_COMPL.SP_WORD75 := W#16#0;
   S711_COMPL.SP_WORD76 := W#16#0;
   S711_COMPL.SP_WORD77 := W#16#0;
   S711_COMPL.SP_WORD78 := W#16#0;
   S711_COMPL.SP_WORD79 := W#16#0;
   S711_COMPL.SP_WORD80 := W#16#0;
   S711_COMPL.SP_WORD81 := W#16#0;
   S711_COMPL.SP_WORD82 := W#16#0;
   S711_COMPL.SP_WORD83 := W#16#0;
   S711_COMPL.SP_WORD84 := W#16#0;
   S711_COMPL.SP_WORD85 := W#16#0;
   S711_COMPL.SP_WORD86 := W#16#0;
   S711_COMPL.SP_WORD87 := W#16#0;
   S711_COMPL.SP_WORD88 := W#16#0;
   S711_COMPL.SP_WORD89 := W#16#0;
   S711_COMPL.SP_WORD90 := W#16#0;
   S711_COMPL.SP_WORD91 := W#16#0;
   S711_COMPL.SP_WORD92 := W#16#0;
   S711_COMPL.SP_WORD93 := W#16#0;
   S711_COMPL.SP_WORD94 := W#16#0;
   S711_COMPL.SP_WORD95 := W#16#0;
   S711_COMPL.SP_WORD96 := W#16#0;
   S711_COMPL.SP_WORD97 := W#16#0;
   S711_COMPL.SP_WORD98 := W#16#0;
   S711_COMPL.SP_WORD99 := W#16#0;
   S711_COMPL.SP_WORD100 := W#16#0;
   S711_COMPL.SP_WORD101 := W#16#0;
END_DATA_BLOCK

DATA_BLOCK DB 53
TITLE =
VERSION : 0.1


  STRUCT
   DISP_CAR_TYPE : STRUCT 	//Temporary placeholder variable
    VIN_NO_1 : WORD ;
    VIN_NO_2 : WORD ;
    CAR_TYPE_1 : WORD ;
    CAR_TYPE_2 : WORD ;
    CAR_TYPE_3 : WORD ;
    CAR_TYPE_4 : WORD ;
    CAR_TYPE_5 : WORD ;
    CAR_TYPE_6 : WORD ;
    RFID_1 : WORD ;
    RFID_2 : WORD ;
   END_STRUCT ;
   WRITE_CAR_TYPE : STRUCT 	//Temporary placeholder variable
    VIN_NO_1 : WORD ;
    VIN_NO_2 : WORD ;
    CAR_TYPE_1 : WORD ;
    CAR_TYPE_2 : WORD ;
    CAR_TYPE_3 : WORD ;
    CAR_TYPE_4 : WORD ;
    CAR_TYPE_5 : WORD ;
    CAR_TYPE_6 : WORD ;
    RFID_1 : WORD ;
    RFID_2 : WORD ;
   END_STRUCT ;
   CAR_TYPE_MODIFY : STRUCT 	//Temporary placeholder variable
    STN_SEL : INT ;
    CCR_ON : BOOL ;
    Modify_ON : BOOL ;
    Car_Type_OK : BOOL ;
    Modify_Set : BOOL ;
    Modify_Reset : BOOL ;
    Modify_Enable : BOOL ;
   END_STRUCT ;
  END_STRUCT ;
BEGIN
   DISP_CAR_TYPE.VIN_NO_1 := W#16#0;
   DISP_CAR_TYPE.VIN_NO_2 := W#16#0;
   DISP_CAR_TYPE.CAR_TYPE_1 := W#16#0;
   DISP_CAR_TYPE.CAR_TYPE_2 := W#16#0;
   DISP_CAR_TYPE.CAR_TYPE_3 := W#16#0;
   DISP_CAR_TYPE.CAR_TYPE_4 := W#16#0;
   DISP_CAR_TYPE.CAR_TYPE_5 := W#16#0;
   DISP_CAR_TYPE.CAR_TYPE_6 := W#16#0;
   DISP_CAR_TYPE.RFID_1 := W#16#0;
   DISP_CAR_TYPE.RFID_2 := W#16#0;
   WRITE_CAR_TYPE.VIN_NO_1 := W#16#0;
   WRITE_CAR_TYPE.VIN_NO_2 := W#16#0;
   WRITE_CAR_TYPE.CAR_TYPE_1 := W#16#0;
   WRITE_CAR_TYPE.CAR_TYPE_2 := W#16#0;
   WRITE_CAR_TYPE.CAR_TYPE_3 := W#16#0;
   WRITE_CAR_TYPE.CAR_TYPE_4 := W#16#0;
   WRITE_CAR_TYPE.CAR_TYPE_5 := W#16#0;
   WRITE_CAR_TYPE.CAR_TYPE_6 := W#16#0;
   WRITE_CAR_TYPE.RFID_1 := W#16#0;
   WRITE_CAR_TYPE.RFID_2 := W#16#0;
   CAR_TYPE_MODIFY.STN_SEL := 0;
   CAR_TYPE_MODIFY.CCR_ON := FALSE;
   CAR_TYPE_MODIFY.Modify_ON := FALSE;
   CAR_TYPE_MODIFY.Car_Type_OK := FALSE;
   CAR_TYPE_MODIFY.Modify_Set := FALSE;
   CAR_TYPE_MODIFY.Modify_Reset := FALSE;
   CAR_TYPE_MODIFY.Modify_Enable := FALSE;
END_DATA_BLOCK

DATA_BLOCK DB 54
TITLE =
VERSION : 0.1


  STRUCT
   DP_1 : STRUCT 	//Temporary placeholder variable
    CHECK_ACTIVE : BOOL ;
    DATA_FIELD : ARRAY  [0 .. 54 ] OF BYTE ;
    SUM_SLAVE_DIAG : INT ;
    LIST_NOT_PRESENT : ARRAY  [0 .. 3 ] OF DWORD ;
    LIST_ERROR : ARRAY  [0 .. 3 ] OF DWORD ;
    RET_VALUE : INT ;
    DIAG_EVENT : BOOL ;
    STATION_ERR : BOOL ;
    RESTART : BOOL ;
    BUSY : BOOL ;
    SP1 : WORD ;
    SP2 : WORD ;
   END_STRUCT ;
   DP_2 : STRUCT 	//Temporary placeholder variable
    CHECK_ACTIVE : BOOL ;
    DATA_FIELD : ARRAY  [0 .. 54 ] OF BYTE ;
    SUM_SLAVE_DIAG : INT ;
    LIST_NOT_PRESENT : ARRAY  [0 .. 3 ] OF DWORD ;
    LIST_ERROR : ARRAY  [0 .. 3 ] OF DWORD ;
    RET_VALUE : INT ;
    DIAG_EVENT : BOOL ;
    STATION_ERR : BOOL ;
    RESTART : BOOL ;
    BUSY : BOOL ;
    SP1 : WORD ;
    SP2 : WORD ;
   END_STRUCT ;
   DP_3 : STRUCT 	//Temporary placeholder variable
    NDR : BOOL ;
    ERR : BOOL ;
    SP21 : ARRAY  [0 .. 3 ] OF WORD ;
    STATUS : WORD ;
    SP22 : WORD ;
    DIAGLNG : BYTE ;
    SP23 : ARRAY  [0 .. 3 ] OF BYTE ;
    LIST_ERROR : ARRAY  [0 .. 3 ] OF DWORD ;
    SP24 : ARRAY  [0 .. 12 ] OF BYTE ;
   END_STRUCT ;
   DP_4 : STRUCT 	//Temporary placeholder variable
    NDR : BOOL ;
    ERR : BOOL ;
    SP21 : ARRAY  [0 .. 3 ] OF WORD ;
    STATUS : WORD ;
    SP22 : WORD ;
    DIAGLNG : BYTE ;
    SP23 : ARRAY  [0 .. 3 ] OF BYTE ;
    LIST_ERROR : ARRAY  [0 .. 3 ] OF DWORD ;
    SP24 : ARRAY  [0 .. 12 ] OF BYTE ;
   END_STRUCT ;
   DP_5 : STRUCT 	//Temporary placeholder variable
    NDR : BOOL ;
    ERR : BOOL ;
    SP21 : ARRAY  [0 .. 3 ] OF WORD ;
    STATUS : WORD ;
    SP22 : WORD ;
    DIAGLNG : BYTE ;
    SP23 : ARRAY  [0 .. 3 ] OF BYTE ;
    LIST_ERROR : ARRAY  [0 .. 3 ] OF DWORD ;
    SP24 : ARRAY  [0 .. 12 ] OF BYTE ;
   END_STRUCT ;
   DP_6 : STRUCT 	//Temporary placeholder variable
    NDR : BOOL ;
    ERR : BOOL ;
    SP21 : ARRAY  [0 .. 3 ] OF WORD ;
    STATUS : WORD ;
    SP22 : WORD ;
    DIAGLNG : BYTE ;
    SP23 : ARRAY  [0 .. 3 ] OF BYTE ;
    LIST_ERROR : ARRAY  [0 .. 3 ] OF DWORD ;
    SP24 : ARRAY  [0 .. 12 ] OF BYTE ;
   END_STRUCT ;
   DP_7 : STRUCT 	//Temporary placeholder variable
    NDR : BOOL ;
    ERR : BOOL ;
    SP21 : ARRAY  [0 .. 3 ] OF WORD ;
    STATUS : WORD ;
    SP22 : WORD ;
    DIAGLNG : BYTE ;
    SP23 : ARRAY  [0 .. 3 ] OF BYTE ;
    LIST_ERROR : ARRAY  [0 .. 3 ] OF DWORD ;
    SP24 : ARRAY  [0 .. 12 ] OF BYTE ;
   END_STRUCT ;
   DP_8 : STRUCT 	//Temporary placeholder variable
    NDR : BOOL ;
    ERR : BOOL ;
    SP21 : ARRAY  [0 .. 3 ] OF WORD ;
    STATUS : WORD ;
    SP22 : WORD ;
    DIAGLNG : BYTE ;
    SP23 : ARRAY  [0 .. 3 ] OF BYTE ;
    LIST_ERROR : ARRAY  [0 .. 3 ] OF DWORD ;
    SP24 : ARRAY  [0 .. 12 ] OF BYTE ;
   END_STRUCT ;
   DP_9 : STRUCT 	//Temporary placeholder variable
    NDR : BOOL ;
    ERR : BOOL ;
    SP21 : ARRAY  [0 .. 3 ] OF WORD ;
    STATUS : WORD ;
    SP22 : WORD ;
    DIAGLNG : BYTE ;
    SP23 : ARRAY  [0 .. 3 ] OF BYTE ;
    LIST_ERROR : ARRAY  [0 .. 3 ] OF DWORD ;
    SP24 : ARRAY  [0 .. 12 ] OF BYTE ;
   END_STRUCT ;
   DP_10 : STRUCT 	//Temporary placeholder variable
    NDR : BOOL ;
    ERR : BOOL ;
    SP21 : ARRAY  [0 .. 3 ] OF WORD ;
    STATUS : WORD ;
    SP22 : WORD ;
    DIAGLNG : BYTE ;
    SP23 : ARRAY  [0 .. 3 ] OF BYTE ;
    LIST_ERROR : ARRAY  [0 .. 3 ] OF DWORD ;
    SP24 : ARRAY  [0 .. 12 ] OF BYTE ;
   END_STRUCT ;
  END_STRUCT ;
BEGIN
   DP_1.CHECK_ACTIVE := FALSE;
   DP_1.DATA_FIELD[0] := B#16#0;
   DP_1.DATA_FIELD[1] := B#16#0;
   DP_1.DATA_FIELD[2] := B#16#0;
   DP_1.DATA_FIELD[3] := B#16#0;
   DP_1.DATA_FIELD[4] := B#16#0;
   DP_1.DATA_FIELD[5] := B#16#0;
   DP_1.DATA_FIELD[6] := B#16#0;
   DP_1.DATA_FIELD[7] := B#16#0;
   DP_1.DATA_FIELD[8] := B#16#0;
   DP_1.DATA_FIELD[9] := B#16#0;
   DP_1.DATA_FIELD[10] := B#16#0;
   DP_1.DATA_FIELD[11] := B#16#0;
   DP_1.DATA_FIELD[12] := B#16#0;
   DP_1.DATA_FIELD[13] := B#16#0;
   DP_1.DATA_FIELD[14] := B#16#0;
   DP_1.DATA_FIELD[15] := B#16#0;
   DP_1.DATA_FIELD[16] := B#16#0;
   DP_1.DATA_FIELD[17] := B#16#0;
   DP_1.DATA_FIELD[18] := B#16#0;
   DP_1.DATA_FIELD[19] := B#16#0;
   DP_1.DATA_FIELD[20] := B#16#0;
   DP_1.DATA_FIELD[21] := B#16#0;
   DP_1.DATA_FIELD[22] := B#16#0;
   DP_1.DATA_FIELD[23] := B#16#0;
   DP_1.DATA_FIELD[24] := B#16#0;
   DP_1.DATA_FIELD[25] := B#16#0;
   DP_1.DATA_FIELD[26] := B#16#0;
   DP_1.DATA_FIELD[27] := B#16#0;
   DP_1.DATA_FIELD[28] := B#16#0;
   DP_1.DATA_FIELD[29] := B#16#0;
   DP_1.DATA_FIELD[30] := B#16#0;
   DP_1.DATA_FIELD[31] := B#16#0;
   DP_1.DATA_FIELD[32] := B#16#0;
   DP_1.DATA_FIELD[33] := B#16#0;
   DP_1.DATA_FIELD[34] := B#16#0;
   DP_1.DATA_FIELD[35] := B#16#0;
   DP_1.DATA_FIELD[36] := B#16#0;
   DP_1.DATA_FIELD[37] := B#16#0;
   DP_1.DATA_FIELD[38] := B#16#0;
   DP_1.DATA_FIELD[39] := B#16#0;
   DP_1.DATA_FIELD[40] := B#16#0;
   DP_1.DATA_FIELD[41] := B#16#0;
   DP_1.DATA_FIELD[42] := B#16#0;
   DP_1.DATA_FIELD[43] := B#16#0;
   DP_1.DATA_FIELD[44] := B#16#0;
   DP_1.DATA_FIELD[45] := B#16#0;
   DP_1.DATA_FIELD[46] := B#16#0;
   DP_1.DATA_FIELD[47] := B#16#0;
   DP_1.DATA_FIELD[48] := B#16#0;
   DP_1.DATA_FIELD[49] := B#16#0;
   DP_1.DATA_FIELD[50] := B#16#0;
   DP_1.DATA_FIELD[51] := B#16#0;
   DP_1.DATA_FIELD[52] := B#16#0;
   DP_1.DATA_FIELD[53] := B#16#0;
   DP_1.DATA_FIELD[54] := B#16#0;
   DP_1.SUM_SLAVE_DIAG := 0;
   DP_1.LIST_NOT_PRESENT[0] := DW#16#0;
   DP_1.LIST_NOT_PRESENT[1] := DW#16#0;
   DP_1.LIST_NOT_PRESENT[2] := DW#16#0;
   DP_1.LIST_NOT_PRESENT[3] := DW#16#0;
   DP_1.LIST_ERROR[0] := DW#16#0;
   DP_1.LIST_ERROR[1] := DW#16#0;
   DP_1.LIST_ERROR[2] := DW#16#0;
   DP_1.LIST_ERROR[3] := DW#16#0;
   DP_1.RET_VALUE := 0;
   DP_1.DIAG_EVENT := FALSE;
   DP_1.STATION_ERR := FALSE;
   DP_1.RESTART := FALSE;
   DP_1.BUSY := FALSE;
   DP_1.SP1 := W#16#0;
   DP_1.SP2 := W#16#0;
   DP_2.CHECK_ACTIVE := FALSE;
   DP_2.DATA_FIELD[0] := B#16#0;
   DP_2.DATA_FIELD[1] := B#16#0;
   DP_2.DATA_FIELD[2] := B#16#0;
   DP_2.DATA_FIELD[3] := B#16#0;
   DP_2.DATA_FIELD[4] := B#16#0;
   DP_2.DATA_FIELD[5] := B#16#0;
   DP_2.DATA_FIELD[6] := B#16#0;
   DP_2.DATA_FIELD[7] := B#16#0;
   DP_2.DATA_FIELD[8] := B#16#0;
   DP_2.DATA_FIELD[9] := B#16#0;
   DP_2.DATA_FIELD[10] := B#16#0;
   DP_2.DATA_FIELD[11] := B#16#0;
   DP_2.DATA_FIELD[12] := B#16#0;
   DP_2.DATA_FIELD[13] := B#16#0;
   DP_2.DATA_FIELD[14] := B#16#0;
   DP_2.DATA_FIELD[15] := B#16#0;
   DP_2.DATA_FIELD[16] := B#16#0;
   DP_2.DATA_FIELD[17] := B#16#0;
   DP_2.DATA_FIELD[18] := B#16#0;
   DP_2.DATA_FIELD[19] := B#16#0;
   DP_2.DATA_FIELD[20] := B#16#0;
   DP_2.DATA_FIELD[21] := B#16#0;
   DP_2.DATA_FIELD[22] := B#16#0;
   DP_2.DATA_FIELD[23] := B#16#0;
   DP_2.DATA_FIELD[24] := B#16#0;
   DP_2.DATA_FIELD[25] := B#16#0;
   DP_2.DATA_FIELD[26] := B#16#0;
   DP_2.DATA_FIELD[27] := B#16#0;
   DP_2.DATA_FIELD[28] := B#16#0;
   DP_2.DATA_FIELD[29] := B#16#0;
   DP_2.DATA_FIELD[30] := B#16#0;
   DP_2.DATA_FIELD[31] := B#16#0;
   DP_2.DATA_FIELD[32] := B#16#0;
   DP_2.DATA_FIELD[33] := B#16#0;
   DP_2.DATA_FIELD[34] := B#16#0;
   DP_2.DATA_FIELD[35] := B#16#0;
   DP_2.DATA_FIELD[36] := B#16#0;
   DP_2.DATA_FIELD[37] := B#16#0;
   DP_2.DATA_FIELD[38] := B#16#0;
   DP_2.DATA_FIELD[39] := B#16#0;
   DP_2.DATA_FIELD[40] := B#16#0;
   DP_2.DATA_FIELD[41] := B#16#0;
   DP_2.DATA_FIELD[42] := B#16#0;
   DP_2.DATA_FIELD[43] := B#16#0;
   DP_2.DATA_FIELD[44] := B#16#0;
   DP_2.DATA_FIELD[45] := B#16#0;
   DP_2.DATA_FIELD[46] := B#16#0;
   DP_2.DATA_FIELD[47] := B#16#0;
   DP_2.DATA_FIELD[48] := B#16#0;
   DP_2.DATA_FIELD[49] := B#16#0;
   DP_2.DATA_FIELD[50] := B#16#0;
   DP_2.DATA_FIELD[51] := B#16#0;
   DP_2.DATA_FIELD[52] := B#16#0;
   DP_2.DATA_FIELD[53] := B#16#0;
   DP_2.DATA_FIELD[54] := B#16#0;
   DP_2.SUM_SLAVE_DIAG := 0;
   DP_2.LIST_NOT_PRESENT[0] := DW#16#0;
   DP_2.LIST_NOT_PRESENT[1] := DW#16#0;
   DP_2.LIST_NOT_PRESENT[2] := DW#16#0;
   DP_2.LIST_NOT_PRESENT[3] := DW#16#0;
   DP_2.LIST_ERROR[0] := DW#16#0;
   DP_2.LIST_ERROR[1] := DW#16#0;
   DP_2.LIST_ERROR[2] := DW#16#0;
   DP_2.LIST_ERROR[3] := DW#16#0;
   DP_2.RET_VALUE := 0;
   DP_2.DIAG_EVENT := FALSE;
   DP_2.STATION_ERR := FALSE;
   DP_2.RESTART := FALSE;
   DP_2.BUSY := FALSE;
   DP_2.SP1 := W#16#0;
   DP_2.SP2 := W#16#0;
   DP_3.NDR := FALSE;
   DP_3.ERR := FALSE;
   DP_3.SP21[0] := W#16#0;
   DP_3.SP21[1] := W#16#0;
   DP_3.SP21[2] := W#16#0;
   DP_3.SP21[3] := W#16#0;
   DP_3.STATUS := W#16#0;
   DP_3.SP22 := W#16#0;
   DP_3.DIAGLNG := B#16#0;
   DP_3.SP23[0] := B#16#0;
   DP_3.SP23[1] := B#16#0;
   DP_3.SP23[2] := B#16#0;
   DP_3.SP23[3] := B#16#0;
   DP_3.LIST_ERROR[0] := DW#16#0;
   DP_3.LIST_ERROR[1] := DW#16#0;
   DP_3.LIST_ERROR[2] := DW#16#0;
   DP_3.LIST_ERROR[3] := DW#16#0;
   DP_3.SP24[0] := B#16#0;
   DP_3.SP24[1] := B#16#0;
   DP_3.SP24[2] := B#16#0;
   DP_3.SP24[3] := B#16#0;
   DP_3.SP24[4] := B#16#0;
   DP_3.SP24[5] := B#16#0;
   DP_3.SP24[6] := B#16#0;
   DP_3.SP24[7] := B#16#0;
   DP_3.SP24[8] := B#16#0;
   DP_3.SP24[9] := B#16#0;
   DP_3.SP24[10] := B#16#0;
   DP_3.SP24[11] := B#16#0;
   DP_3.SP24[12] := B#16#0;
   DP_4.NDR := FALSE;
   DP_4.ERR := FALSE;
   DP_4.SP21[0] := W#16#0;
   DP_4.SP21[1] := W#16#0;
   DP_4.SP21[2] := W#16#0;
   DP_4.SP21[3] := W#16#0;
   DP_4.STATUS := W#16#0;
   DP_4.SP22 := W#16#0;
   DP_4.DIAGLNG := B#16#0;
   DP_4.SP23[0] := B#16#0;
   DP_4.SP23[1] := B#16#0;
   DP_4.SP23[2] := B#16#0;
   DP_4.SP23[3] := B#16#0;
   DP_4.LIST_ERROR[0] := DW#16#0;
   DP_4.LIST_ERROR[1] := DW#16#0;
   DP_4.LIST_ERROR[2] := DW#16#0;
   DP_4.LIST_ERROR[3] := DW#16#0;
   DP_4.SP24[0] := B#16#0;
   DP_4.SP24[1] := B#16#0;
   DP_4.SP24[2] := B#16#0;
   DP_4.SP24[3] := B#16#0;
   DP_4.SP24[4] := B#16#0;
   DP_4.SP24[5] := B#16#0;
   DP_4.SP24[6] := B#16#0;
   DP_4.SP24[7] := B#16#0;
   DP_4.SP24[8] := B#16#0;
   DP_4.SP24[9] := B#16#0;
   DP_4.SP24[10] := B#16#0;
   DP_4.SP24[11] := B#16#0;
   DP_4.SP24[12] := B#16#0;
   DP_5.NDR := FALSE;
   DP_5.ERR := FALSE;
   DP_5.SP21[0] := W#16#0;
   DP_5.SP21[1] := W#16#0;
   DP_5.SP21[2] := W#16#0;
   DP_5.SP21[3] := W#16#0;
   DP_5.STATUS := W#16#0;
   DP_5.SP22 := W#16#0;
   DP_5.DIAGLNG := B#16#0;
   DP_5.SP23[0] := B#16#0;
   DP_5.SP23[1] := B#16#0;
   DP_5.SP23[2] := B#16#0;
   DP_5.SP23[3] := B#16#0;
   DP_5.LIST_ERROR[0] := DW#16#0;
   DP_5.LIST_ERROR[1] := DW#16#0;
   DP_5.LIST_ERROR[2] := DW#16#0;
   DP_5.LIST_ERROR[3] := DW#16#0;
   DP_5.SP24[0] := B#16#0;
   DP_5.SP24[1] := B#16#0;
   DP_5.SP24[2] := B#16#0;
   DP_5.SP24[3] := B#16#0;
   DP_5.SP24[4] := B#16#0;
   DP_5.SP24[5] := B#16#0;
   DP_5.SP24[6] := B#16#0;
   DP_5.SP24[7] := B#16#0;
   DP_5.SP24[8] := B#16#0;
   DP_5.SP24[9] := B#16#0;
   DP_5.SP24[10] := B#16#0;
   DP_5.SP24[11] := B#16#0;
   DP_5.SP24[12] := B#16#0;
   DP_6.NDR := FALSE;
   DP_6.ERR := FALSE;
   DP_6.SP21[0] := W#16#0;
   DP_6.SP21[1] := W#16#0;
   DP_6.SP21[2] := W#16#0;
   DP_6.SP21[3] := W#16#0;
   DP_6.STATUS := W#16#0;
   DP_6.SP22 := W#16#0;
   DP_6.DIAGLNG := B#16#0;
   DP_6.SP23[0] := B#16#0;
   DP_6.SP23[1] := B#16#0;
   DP_6.SP23[2] := B#16#0;
   DP_6.SP23[3] := B#16#0;
   DP_6.LIST_ERROR[0] := DW#16#0;
   DP_6.LIST_ERROR[1] := DW#16#0;
   DP_6.LIST_ERROR[2] := DW#16#0;
   DP_6.LIST_ERROR[3] := DW#16#0;
   DP_6.SP24[0] := B#16#0;
   DP_6.SP24[1] := B#16#0;
   DP_6.SP24[2] := B#16#0;
   DP_6.SP24[3] := B#16#0;
   DP_6.SP24[4] := B#16#0;
   DP_6.SP24[5] := B#16#0;
   DP_6.SP24[6] := B#16#0;
   DP_6.SP24[7] := B#16#0;
   DP_6.SP24[8] := B#16#0;
   DP_6.SP24[9] := B#16#0;
   DP_6.SP24[10] := B#16#0;
   DP_6.SP24[11] := B#16#0;
   DP_6.SP24[12] := B#16#0;
   DP_7.NDR := FALSE;
   DP_7.ERR := FALSE;
   DP_7.SP21[0] := W#16#0;
   DP_7.SP21[1] := W#16#0;
   DP_7.SP21[2] := W#16#0;
   DP_7.SP21[3] := W#16#0;
   DP_7.STATUS := W#16#0;
   DP_7.SP22 := W#16#0;
   DP_7.DIAGLNG := B#16#0;
   DP_7.SP23[0] := B#16#0;
   DP_7.SP23[1] := B#16#0;
   DP_7.SP23[2] := B#16#0;
   DP_7.SP23[3] := B#16#0;
   DP_7.LIST_ERROR[0] := DW#16#0;
   DP_7.LIST_ERROR[1] := DW#16#0;
   DP_7.LIST_ERROR[2] := DW#16#0;
   DP_7.LIST_ERROR[3] := DW#16#0;
   DP_7.SP24[0] := B#16#0;
   DP_7.SP24[1] := B#16#0;
   DP_7.SP24[2] := B#16#0;
   DP_7.SP24[3] := B#16#0;
   DP_7.SP24[4] := B#16#0;
   DP_7.SP24[5] := B#16#0;
   DP_7.SP24[6] := B#16#0;
   DP_7.SP24[7] := B#16#0;
   DP_7.SP24[8] := B#16#0;
   DP_7.SP24[9] := B#16#0;
   DP_7.SP24[10] := B#16#0;
   DP_7.SP24[11] := B#16#0;
   DP_7.SP24[12] := B#16#0;
   DP_8.NDR := FALSE;
   DP_8.ERR := FALSE;
   DP_8.SP21[0] := W#16#0;
   DP_8.SP21[1] := W#16#0;
   DP_8.SP21[2] := W#16#0;
   DP_8.SP21[3] := W#16#0;
   DP_8.STATUS := W#16#0;
   DP_8.SP22 := W#16#0;
   DP_8.DIAGLNG := B#16#0;
   DP_8.SP23[0] := B#16#0;
   DP_8.SP23[1] := B#16#0;
   DP_8.SP23[2] := B#16#0;
   DP_8.SP23[3] := B#16#0;
   DP_8.LIST_ERROR[0] := DW#16#0;
   DP_8.LIST_ERROR[1] := DW#16#0;
   DP_8.LIST_ERROR[2] := DW#16#0;
   DP_8.LIST_ERROR[3] := DW#16#0;
   DP_8.SP24[0] := B#16#0;
   DP_8.SP24[1] := B#16#0;
   DP_8.SP24[2] := B#16#0;
   DP_8.SP24[3] := B#16#0;
   DP_8.SP24[4] := B#16#0;
   DP_8.SP24[5] := B#16#0;
   DP_8.SP24[6] := B#16#0;
   DP_8.SP24[7] := B#16#0;
   DP_8.SP24[8] := B#16#0;
   DP_8.SP24[9] := B#16#0;
   DP_8.SP24[10] := B#16#0;
   DP_8.SP24[11] := B#16#0;
   DP_8.SP24[12] := B#16#0;
   DP_9.NDR := FALSE;
   DP_9.ERR := FALSE;
   DP_9.SP21[0] := W#16#0;
   DP_9.SP21[1] := W#16#0;
   DP_9.SP21[2] := W#16#0;
   DP_9.SP21[3] := W#16#0;
   DP_9.STATUS := W#16#0;
   DP_9.SP22 := W#16#0;
   DP_9.DIAGLNG := B#16#0;
   DP_9.SP23[0] := B#16#0;
   DP_9.SP23[1] := B#16#0;
   DP_9.SP23[2] := B#16#0;
   DP_9.SP23[3] := B#16#0;
   DP_9.LIST_ERROR[0] := DW#16#0;
   DP_9.LIST_ERROR[1] := DW#16#0;
   DP_9.LIST_ERROR[2] := DW#16#0;
   DP_9.LIST_ERROR[3] := DW#16#0;
   DP_9.SP24[0] := B#16#0;
   DP_9.SP24[1] := B#16#0;
   DP_9.SP24[2] := B#16#0;
   DP_9.SP24[3] := B#16#0;
   DP_9.SP24[4] := B#16#0;
   DP_9.SP24[5] := B#16#0;
   DP_9.SP24[6] := B#16#0;
   DP_9.SP24[7] := B#16#0;
   DP_9.SP24[8] := B#16#0;
   DP_9.SP24[9] := B#16#0;
   DP_9.SP24[10] := B#16#0;
   DP_9.SP24[11] := B#16#0;
   DP_9.SP24[12] := B#16#0;
   DP_10.NDR := FALSE;
   DP_10.ERR := FALSE;
   DP_10.SP21[0] := W#16#0;
   DP_10.SP21[1] := W#16#0;
   DP_10.SP21[2] := W#16#0;
   DP_10.SP21[3] := W#16#0;
   DP_10.STATUS := W#16#0;
   DP_10.SP22 := W#16#0;
   DP_10.DIAGLNG := B#16#0;
   DP_10.SP23[0] := B#16#0;
   DP_10.SP23[1] := B#16#0;
   DP_10.SP23[2] := B#16#0;
   DP_10.SP23[3] := B#16#0;
   DP_10.LIST_ERROR[0] := DW#16#0;
   DP_10.LIST_ERROR[1] := DW#16#0;
   DP_10.LIST_ERROR[2] := DW#16#0;
   DP_10.LIST_ERROR[3] := DW#16#0;
   DP_10.SP24[0] := B#16#0;
   DP_10.SP24[1] := B#16#0;
   DP_10.SP24[2] := B#16#0;
   DP_10.SP24[3] := B#16#0;
   DP_10.SP24[4] := B#16#0;
   DP_10.SP24[5] := B#16#0;
   DP_10.SP24[6] := B#16#0;
   DP_10.SP24[7] := B#16#0;
   DP_10.SP24[8] := B#16#0;
   DP_10.SP24[9] := B#16#0;
   DP_10.SP24[10] := B#16#0;
   DP_10.SP24[11] := B#16#0;
   DP_10.SP24[12] := B#16#0;
END_DATA_BLOCK

DATA_BLOCK DB 55
TITLE =
VERSION : 0.1


  STRUCT
   CP1 : STRUCT
    FC2_NDR : BOOL ;
    FC2_ERROR : BOOL ;
    SP1 : BOOL ;
    SP2 : BOOL ;
    FC1_NDR : BOOL ;
    FC1_ERROR : BOOL ;
    SP3 : BOOL ;
    SP4 : BOOL ;
    FC2_STATUS : WORD ;
    FC2_DPSTATUS : BYTE ;
    FC1_STATUS : WORD ;
    SP5 : WORD ;
    SFC20_1_RET_VAL : INT ;
    SFC20_2_RET_VAL : INT ;
    SFC20_3_RET_VAL : INT ;
    SFC20_4_RET_VAL : INT ;
    SFC20_5_RET_VAL : INT ;
    SFC20_6_RET_VAL : INT ;
    SFC20_7_RET_VAL : INT ;
    SFC20_8_RET_VAL : INT ;
    SFC20_9_RET_VAL : INT ;
    SFC20_10_RET_VAL : INT ;
    SP : ARRAY  [0 .. 9 ] OF WORD ;
   END_STRUCT ;
   CP2 : STRUCT
    FC2_NDR : BOOL ;
    FC2_ERROR : BOOL ;
    SP1 : BOOL ;
    SP2 : BOOL ;
    FC1_NDR : BOOL ;
    FC1_ERROR : BOOL ;
    SP3 : BOOL ;
    SP4 : BOOL ;
    FC2_STATUS : WORD ;
    FC2_DPSTATUS : BYTE ;
    FC1_STATUS : WORD ;
    SP5 : WORD ;
    SFC20_1_RET_VAL : INT ;
    SFC20_2_RET_VAL : INT ;
    SFC20_3_RET_VAL : INT ;
    SFC20_4_RET_VAL : INT ;
    SFC20_5_RET_VAL : INT ;
    SFC20_6_RET_VAL : INT ;
    SFC20_7_RET_VAL : INT ;
    SFC20_8_RET_VAL : INT ;
    SFC20_9_RET_VAL : INT ;
    SFC20_10_RET_VAL : INT ;
    SP : ARRAY  [0 .. 9 ] OF WORD ;
   END_STRUCT ;
   CP3 : STRUCT
    FC2_NDR : BOOL ;
    FC2_ERROR : BOOL ;
    SP1 : BOOL ;
    SP2 : BOOL ;
    FC1_NDR : BOOL ;
    FC1_ERROR : BOOL ;
    SP3 : BOOL ;
    SP4 : BOOL ;
    FC2_STATUS : WORD ;
    FC2_DPSTATUS : BYTE ;
    FC1_STATUS : WORD ;
    SP5 : WORD ;
    SFC20_1_RET_VAL : INT ;
    SFC20_2_RET_VAL : INT ;
    SFC20_3_RET_VAL : INT ;
    SFC20_4_RET_VAL : INT ;
    SFC20_5_RET_VAL : INT ;
    SFC20_6_RET_VAL : INT ;
    SFC20_7_RET_VAL : INT ;
    SFC20_8_RET_VAL : INT ;
    SFC20_9_RET_VAL : INT ;
    SFC20_10_RET_VAL : INT ;
    SP : ARRAY  [0 .. 9 ] OF WORD ;
   END_STRUCT ;
   CP4 : STRUCT
    FC2_NDR : BOOL ;
    FC2_ERROR : BOOL ;
    SP1 : BOOL ;
    SP2 : BOOL ;
    FC1_NDR : BOOL ;
    FC1_ERROR : BOOL ;
    SP3 : BOOL ;
    SP4 : BOOL ;
    FC2_STATUS : WORD ;
    FC2_DPSTATUS : BYTE ;
    FC1_STATUS : WORD ;
    SP5 : WORD ;
    SFC20_1_RET_VAL : INT ;
    SFC20_2_RET_VAL : INT ;
    SFC20_3_RET_VAL : INT ;
    SFC20_4_RET_VAL : INT ;
    SFC20_5_RET_VAL : INT ;
    SFC20_6_RET_VAL : INT ;
    SFC20_7_RET_VAL : INT ;
    SFC20_8_RET_VAL : INT ;
    SFC20_9_RET_VAL : INT ;
    SFC20_10_RET_VAL : INT ;
    SP : ARRAY  [0 .. 9 ] OF WORD ;
   END_STRUCT ;
   CP5 : STRUCT
    FC2_NDR : BOOL ;
    FC2_ERROR : BOOL ;
    SP1 : BOOL ;
    SP2 : BOOL ;
    FC1_NDR : BOOL ;
    FC1_ERROR : BOOL ;
    SP3 : BOOL ;
    SP4 : BOOL ;
    FC2_STATUS : WORD ;
    FC2_DPSTATUS : BYTE ;
    FC1_STATUS : WORD ;
    SP5 : WORD ;
    SFC20_1_RET_VAL : INT ;
    SFC20_2_RET_VAL : INT ;
    SFC20_3_RET_VAL : INT ;
    SFC20_4_RET_VAL : INT ;
    SFC20_5_RET_VAL : INT ;
    SFC20_6_RET_VAL : INT ;
    SFC20_7_RET_VAL : INT ;
    SFC20_8_RET_VAL : INT ;
    SFC20_9_RET_VAL : INT ;
    SFC20_10_RET_VAL : INT ;
    SP : ARRAY  [0 .. 9 ] OF WORD ;
   END_STRUCT ;
   CP6 : STRUCT
    FC2_NDR : BOOL ;
    FC2_ERROR : BOOL ;
    SP1 : BOOL ;
    SP2 : BOOL ;
    FC1_NDR : BOOL ;
    FC1_ERROR : BOOL ;
    SP3 : BOOL ;
    SP4 : BOOL ;
    FC2_STATUS : WORD ;
    FC2_DPSTATUS : BYTE ;
    FC1_STATUS : WORD ;
    SP5 : WORD ;
    SFC20_1_RET_VAL : INT ;
    SFC20_2_RET_VAL : INT ;
    SFC20_3_RET_VAL : INT ;
    SFC20_4_RET_VAL : INT ;
    SFC20_5_RET_VAL : INT ;
    SFC20_6_RET_VAL : INT ;
    SFC20_7_RET_VAL : INT ;
    SFC20_8_RET_VAL : INT ;
    SFC20_9_RET_VAL : INT ;
    SFC20_10_RET_VAL : INT ;
    SP : ARRAY  [0 .. 9 ] OF WORD ;
   END_STRUCT ;
   CP7 : STRUCT
    FC2_NDR : BOOL ;
    FC2_ERROR : BOOL ;
    SP1 : BOOL ;
    SP2 : BOOL ;
    FC1_NDR : BOOL ;
    FC1_ERROR : BOOL ;
    SP3 : BOOL ;
    SP4 : BOOL ;
    FC2_STATUS : WORD ;
    FC2_DPSTATUS : BYTE ;
    FC1_STATUS : WORD ;
    SP5 : WORD ;
    SFC20_1_RET_VAL : INT ;
    SFC20_2_RET_VAL : INT ;
    SFC20_3_RET_VAL : INT ;
    SFC20_4_RET_VAL : INT ;
    SFC20_5_RET_VAL : INT ;
    SFC20_6_RET_VAL : INT ;
    SFC20_7_RET_VAL : INT ;
    SFC20_8_RET_VAL : INT ;
    SFC20_9_RET_VAL : INT ;
    SFC20_10_RET_VAL : INT ;
    SP : ARRAY  [0 .. 9 ] OF WORD ;
   END_STRUCT ;
   CP8 : STRUCT
    FC2_NDR : BOOL ;
    FC2_ERROR : BOOL ;
    SP1 : BOOL ;
    SP2 : BOOL ;
    FC1_NDR : BOOL ;
    FC1_ERROR : BOOL ;
    SP3 : BOOL ;
    SP4 : BOOL ;
    FC2_STATUS : WORD ;
    FC2_DPSTATUS : BYTE ;
    FC1_STATUS : WORD ;
    SP5 : WORD ;
    SFC20_1_RET_VAL : INT ;
    SFC20_2_RET_VAL : INT ;
    SFC20_3_RET_VAL : INT ;
    SFC20_4_RET_VAL : INT ;
    SFC20_5_RET_VAL : INT ;
    SFC20_6_RET_VAL : INT ;
    SFC20_7_RET_VAL : INT ;
    SFC20_8_RET_VAL : INT ;
    SFC20_9_RET_VAL : INT ;
    SFC20_10_RET_VAL : INT ;
    SP : ARRAY  [0 .. 9 ] OF WORD ;
   END_STRUCT ;
   RTN_VALUE_WORD : ARRAY  [0 .. 49 ] OF WORD ;
   AG1 : STRUCT
    FC6_NDR : BOOL ;
    FC6_ERROR : BOOL ;
    SP1 : BOOL ;
    SP2 : BOOL ;
    FC5_NDR : BOOL ;
    FC5_ERROR : BOOL ;
    SP3 : BOOL ;
    SP4 : BOOL ;
    FC6_STATUS : WORD ;
    FC6_DPSTATUS : BYTE ;
    FC5_STATUS : WORD ;
    SP5 : WORD ;
    SFC20_1_RET_VAL : INT ;
    SFC20_2_RET_VAL : INT ;
    SFC20_3_RET_VAL : INT ;
    SFC20_4_RET_VAL : INT ;
    SFC20_5_RET_VAL : INT ;
    SFC20_6_RET_VAL : INT ;
    SFC20_7_RET_VAL : INT ;
    SFC20_8_RET_VAL : INT ;
    SFC20_9_RET_VAL : INT ;
    SFC20_10_RET_VAL : INT ;
    SP : ARRAY  [0 .. 9 ] OF WORD ;
   END_STRUCT ;
   AG2 : STRUCT
    FC6_NDR : BOOL ;
    FC6_ERROR : BOOL ;
    SP1 : BOOL ;
    SP2 : BOOL ;
    FC5_NDR : BOOL ;
    FC5_ERROR : BOOL ;
    SP3 : BOOL ;
    SP4 : BOOL ;
    FC6_STATUS : WORD ;
    FC6_DPSTATUS : BYTE ;
    FC5_STATUS : WORD ;
    SP5 : WORD ;
    SFC20_1_RET_VAL : INT ;
    SFC20_2_RET_VAL : INT ;
    SFC20_3_RET_VAL : INT ;
    SFC20_4_RET_VAL : INT ;
    SFC20_5_RET_VAL : INT ;
    SFC20_6_RET_VAL : INT ;
    SFC20_7_RET_VAL : INT ;
    SFC20_8_RET_VAL : INT ;
    SFC20_9_RET_VAL : INT ;
    SFC20_10_RET_VAL : INT ;
    SP : ARRAY  [0 .. 9 ] OF WORD ;
   END_STRUCT ;
   AG3 : STRUCT
    FC6_NDR : BOOL ;
    FC6_ERROR : BOOL ;
    SP1 : BOOL ;
    SP2 : BOOL ;
    FC5_NDR : BOOL ;
    FC5_ERROR : BOOL ;
    SP3 : BOOL ;
    SP4 : BOOL ;
    FC6_STATUS : WORD ;
    FC6_DPSTATUS : BYTE ;
    FC5_STATUS : WORD ;
    SP5 : WORD ;
    SFC20_1_RET_VAL : INT ;
    SFC20_2_RET_VAL : INT ;
    SFC20_3_RET_VAL : INT ;
    SFC20_4_RET_VAL : INT ;
    SFC20_5_RET_VAL : INT ;
    SFC20_6_RET_VAL : INT ;
    SFC20_7_RET_VAL : INT ;
    SFC20_8_RET_VAL : INT ;
    SFC20_9_RET_VAL : INT ;
    SFC20_10_RET_VAL : INT ;
    SP : ARRAY  [0 .. 9 ] OF WORD ;
   END_STRUCT ;
   AG4 : STRUCT
    FC6_NDR : BOOL ;
    FC6_ERROR : BOOL ;
    SP1 : BOOL ;
    SP2 : BOOL ;
    FC5_NDR : BOOL ;
    FC5_ERROR : BOOL ;
    SP3 : BOOL ;
    SP4 : BOOL ;
    FC6_STATUS : WORD ;
    FC6_DPSTATUS : BYTE ;
    FC5_STATUS : WORD ;
    SP5 : WORD ;
    SFC20_1_RET_VAL : INT ;
    SFC20_2_RET_VAL : INT ;
    SFC20_3_RET_VAL : INT ;
    SFC20_4_RET_VAL : INT ;
    SFC20_5_RET_VAL : INT ;
    SFC20_6_RET_VAL : INT ;
    SFC20_7_RET_VAL : INT ;
    SFC20_8_RET_VAL : INT ;
    SFC20_9_RET_VAL : INT ;
    SFC20_10_RET_VAL : INT ;
    SP : ARRAY  [0 .. 9 ] OF WORD ;
   END_STRUCT ;
   AG5 : STRUCT
    FC6_NDR : BOOL ;
    FC6_ERROR : BOOL ;
    SP1 : BOOL ;
    SP2 : BOOL ;
    FC5_NDR : BOOL ;
    FC5_ERROR : BOOL ;
    SP3 : BOOL ;
    SP4 : BOOL ;
    FC6_STATUS : WORD ;
    FC6_DPSTATUS : BYTE ;
    FC5_STATUS : WORD ;
    SP5 : WORD ;
    SFC20_1_RET_VAL : INT ;
    SFC20_2_RET_VAL : INT ;
    SFC20_3_RET_VAL : INT ;
    SFC20_4_RET_VAL : INT ;
    SFC20_5_RET_VAL : INT ;
    SFC20_6_RET_VAL : INT ;
    SFC20_7_RET_VAL : INT ;
    SFC20_8_RET_VAL : INT ;
    SFC20_9_RET_VAL : INT ;
    SFC20_10_RET_VAL : INT ;
    SP : ARRAY  [0 .. 9 ] OF WORD ;
   END_STRUCT ;
   AG6 : STRUCT
    FC6_NDR : BOOL ;
    FC6_ERROR : BOOL ;
    SP1 : BOOL ;
    SP2 : BOOL ;
    FC5_NDR : BOOL ;
    FC5_ERROR : BOOL ;
    SP3 : BOOL ;
    SP4 : BOOL ;
    FC6_STATUS : WORD ;
    FC6_DPSTATUS : BYTE ;
    FC5_STATUS : WORD ;
    SP5 : WORD ;
    SFC20_1_RET_VAL : INT ;
    SFC20_2_RET_VAL : INT ;
    SFC20_3_RET_VAL : INT ;
    SFC20_4_RET_VAL : INT ;
    SFC20_5_RET_VAL : INT ;
    SFC20_6_RET_VAL : INT ;
    SFC20_7_RET_VAL : INT ;
    SFC20_8_RET_VAL : INT ;
    SFC20_9_RET_VAL : INT ;
    SFC20_10_RET_VAL : INT ;
    SP : ARRAY  [0 .. 9 ] OF WORD ;
   END_STRUCT ;
   AG7 : STRUCT
    FC6_NDR : BOOL ;
    FC6_ERROR : BOOL ;
    SP1 : BOOL ;
    SP2 : BOOL ;
    FC5_NDR : BOOL ;
    FC5_ERROR : BOOL ;
    SP3 : BOOL ;
    SP4 : BOOL ;
    FC6_STATUS : WORD ;
    FC6_DPSTATUS : BYTE ;
    FC5_STATUS : WORD ;
    SP5 : WORD ;
    SFC20_1_RET_VAL : INT ;
    SFC20_2_RET_VAL : INT ;
    SFC20_3_RET_VAL : INT ;
    SFC20_4_RET_VAL : INT ;
    SFC20_5_RET_VAL : INT ;
    SFC20_6_RET_VAL : INT ;
    SFC20_7_RET_VAL : INT ;
    SFC20_8_RET_VAL : INT ;
    SFC20_9_RET_VAL : INT ;
    SFC20_10_RET_VAL : INT ;
    SP : ARRAY  [0 .. 9 ] OF WORD ;
   END_STRUCT ;
   SP : ARRAY  [0 .. 74 ] OF WORD ;
   CTYPE_RET_VAL : ARRAY  [0 .. 99 ] OF INT ;
   MES_RET_VAL1 : ARRAY  [0 .. 199 ] OF INT ;
  END_STRUCT ;
BEGIN
   CP1.FC2_NDR := FALSE;
   CP1.FC2_ERROR := FALSE;
   CP1.SP1 := FALSE;
   CP1.SP2 := FALSE;
   CP1.FC1_NDR := FALSE;
   CP1.FC1_ERROR := FALSE;
   CP1.SP3 := FALSE;
   CP1.SP4 := FALSE;
   CP1.FC2_STATUS := W#16#0;
   CP1.FC2_DPSTATUS := B#16#0;
   CP1.FC1_STATUS := W#16#0;
   CP1.SP5 := W#16#0;
   CP1.SFC20_1_RET_VAL := 0;
   CP1.SFC20_2_RET_VAL := 0;
   CP1.SFC20_3_RET_VAL := 0;
   CP1.SFC20_4_RET_VAL := 0;
   CP1.SFC20_5_RET_VAL := 0;
   CP1.SFC20_6_RET_VAL := 0;
   CP1.SFC20_7_RET_VAL := 0;
   CP1.SFC20_8_RET_VAL := 0;
   CP1.SFC20_9_RET_VAL := 0;
   CP1.SFC20_10_RET_VAL := 0;
   CP1.SP[0] := W#16#0;
   CP1.SP[1] := W#16#0;
   CP1.SP[2] := W#16#0;
   CP1.SP[3] := W#16#0;
   CP1.SP[4] := W#16#0;
   CP1.SP[5] := W#16#0;
   CP1.SP[6] := W#16#0;
   CP1.SP[7] := W#16#0;
   CP1.SP[8] := W#16#0;
   CP1.SP[9] := W#16#0;
   CP2.FC2_NDR := FALSE;
   CP2.FC2_ERROR := FALSE;
   CP2.SP1 := FALSE;
   CP2.SP2 := FALSE;
   CP2.FC1_NDR := FALSE;
   CP2.FC1_ERROR := FALSE;
   CP2.SP3 := FALSE;
   CP2.SP4 := FALSE;
   CP2.FC2_STATUS := W#16#0;
   CP2.FC2_DPSTATUS := B#16#0;
   CP2.FC1_STATUS := W#16#0;
   CP2.SP5 := W#16#0;
   CP2.SFC20_1_RET_VAL := 0;
   CP2.SFC20_2_RET_VAL := 0;
   CP2.SFC20_3_RET_VAL := 0;
   CP2.SFC20_4_RET_VAL := 0;
   CP2.SFC20_5_RET_VAL := 0;
   CP2.SFC20_6_RET_VAL := 0;
   CP2.SFC20_7_RET_VAL := 0;
   CP2.SFC20_8_RET_VAL := 0;
   CP2.SFC20_9_RET_VAL := 0;
   CP2.SFC20_10_RET_VAL := 0;
   CP2.SP[0] := W#16#0;
   CP2.SP[1] := W#16#0;
   CP2.SP[2] := W#16#0;
   CP2.SP[3] := W#16#0;
   CP2.SP[4] := W#16#0;
   CP2.SP[5] := W#16#0;
   CP2.SP[6] := W#16#0;
   CP2.SP[7] := W#16#0;
   CP2.SP[8] := W#16#0;
   CP2.SP[9] := W#16#0;
   CP3.FC2_NDR := FALSE;
   CP3.FC2_ERROR := FALSE;
   CP3.SP1 := FALSE;
   CP3.SP2 := FALSE;
   CP3.FC1_NDR := FALSE;
   CP3.FC1_ERROR := FALSE;
   CP3.SP3 := FALSE;
   CP3.SP4 := FALSE;
   CP3.FC2_STATUS := W#16#0;
   CP3.FC2_DPSTATUS := B#16#0;
   CP3.FC1_STATUS := W#16#0;
   CP3.SP5 := W#16#0;
   CP3.SFC20_1_RET_VAL := 0;
   CP3.SFC20_2_RET_VAL := 0;
   CP3.SFC20_3_RET_VAL := 0;
   CP3.SFC20_4_RET_VAL := 0;
   CP3.SFC20_5_RET_VAL := 0;
   CP3.SFC20_6_RET_VAL := 0;
   CP3.SFC20_7_RET_VAL := 0;
   CP3.SFC20_8_RET_VAL := 0;
   CP3.SFC20_9_RET_VAL := 0;
   CP3.SFC20_10_RET_VAL := 0;
   CP3.SP[0] := W#16#0;
   CP3.SP[1] := W#16#0;
   CP3.SP[2] := W#16#0;
   CP3.SP[3] := W#16#0;
   CP3.SP[4] := W#16#0;
   CP3.SP[5] := W#16#0;
   CP3.SP[6] := W#16#0;
   CP3.SP[7] := W#16#0;
   CP3.SP[8] := W#16#0;
   CP3.SP[9] := W#16#0;
   CP4.FC2_NDR := FALSE;
   CP4.FC2_ERROR := FALSE;
   CP4.SP1 := FALSE;
   CP4.SP2 := FALSE;
   CP4.FC1_NDR := FALSE;
   CP4.FC1_ERROR := FALSE;
   CP4.SP3 := FALSE;
   CP4.SP4 := FALSE;
   CP4.FC2_STATUS := W#16#0;
   CP4.FC2_DPSTATUS := B#16#0;
   CP4.FC1_STATUS := W#16#0;
   CP4.SP5 := W#16#0;
   CP4.SFC20_1_RET_VAL := 0;
   CP4.SFC20_2_RET_VAL := 0;
   CP4.SFC20_3_RET_VAL := 0;
   CP4.SFC20_4_RET_VAL := 0;
   CP4.SFC20_5_RET_VAL := 0;
   CP4.SFC20_6_RET_VAL := 0;
   CP4.SFC20_7_RET_VAL := 0;
   CP4.SFC20_8_RET_VAL := 0;
   CP4.SFC20_9_RET_VAL := 0;
   CP4.SFC20_10_RET_VAL := 0;
   CP4.SP[0] := W#16#0;
   CP4.SP[1] := W#16#0;
   CP4.SP[2] := W#16#0;
   CP4.SP[3] := W#16#0;
   CP4.SP[4] := W#16#0;
   CP4.SP[5] := W#16#0;
   CP4.SP[6] := W#16#0;
   CP4.SP[7] := W#16#0;
   CP4.SP[8] := W#16#0;
   CP4.SP[9] := W#16#0;
   CP5.FC2_NDR := FALSE;
   CP5.FC2_ERROR := FALSE;
   CP5.SP1 := FALSE;
   CP5.SP2 := FALSE;
   CP5.FC1_NDR := FALSE;
   CP5.FC1_ERROR := FALSE;
   CP5.SP3 := FALSE;
   CP5.SP4 := FALSE;
   CP5.FC2_STATUS := W#16#0;
   CP5.FC2_DPSTATUS := B#16#0;
   CP5.FC1_STATUS := W#16#0;
   CP5.SP5 := W#16#0;
   CP5.SFC20_1_RET_VAL := 0;
   CP5.SFC20_2_RET_VAL := 0;
   CP5.SFC20_3_RET_VAL := 0;
   CP5.SFC20_4_RET_VAL := 0;
   CP5.SFC20_5_RET_VAL := 0;
   CP5.SFC20_6_RET_VAL := 0;
   CP5.SFC20_7_RET_VAL := 0;
   CP5.SFC20_8_RET_VAL := 0;
   CP5.SFC20_9_RET_VAL := 0;
   CP5.SFC20_10_RET_VAL := 0;
   CP5.SP[0] := W#16#0;
   CP5.SP[1] := W#16#0;
   CP5.SP[2] := W#16#0;
   CP5.SP[3] := W#16#0;
   CP5.SP[4] := W#16#0;
   CP5.SP[5] := W#16#0;
   CP5.SP[6] := W#16#0;
   CP5.SP[7] := W#16#0;
   CP5.SP[8] := W#16#0;
   CP5.SP[9] := W#16#0;
   CP6.FC2_NDR := FALSE;
   CP6.FC2_ERROR := FALSE;
   CP6.SP1 := FALSE;
   CP6.SP2 := FALSE;
   CP6.FC1_NDR := FALSE;
   CP6.FC1_ERROR := FALSE;
   CP6.SP3 := FALSE;
   CP6.SP4 := FALSE;
   CP6.FC2_STATUS := W#16#0;
   CP6.FC2_DPSTATUS := B#16#0;
   CP6.FC1_STATUS := W#16#0;
   CP6.SP5 := W#16#0;
   CP6.SFC20_1_RET_VAL := 0;
   CP6.SFC20_2_RET_VAL := 0;
   CP6.SFC20_3_RET_VAL := 0;
   CP6.SFC20_4_RET_VAL := 0;
   CP6.SFC20_5_RET_VAL := 0;
   CP6.SFC20_6_RET_VAL := 0;
   CP6.SFC20_7_RET_VAL := 0;
   CP6.SFC20_8_RET_VAL := 0;
   CP6.SFC20_9_RET_VAL := 0;
   CP6.SFC20_10_RET_VAL := 0;
   CP6.SP[0] := W#16#0;
   CP6.SP[1] := W#16#0;
   CP6.SP[2] := W#16#0;
   CP6.SP[3] := W#16#0;
   CP6.SP[4] := W#16#0;
   CP6.SP[5] := W#16#0;
   CP6.SP[6] := W#16#0;
   CP6.SP[7] := W#16#0;
   CP6.SP[8] := W#16#0;
   CP6.SP[9] := W#16#0;
   CP7.FC2_NDR := FALSE;
   CP7.FC2_ERROR := FALSE;
   CP7.SP1 := FALSE;
   CP7.SP2 := FALSE;
   CP7.FC1_NDR := FALSE;
   CP7.FC1_ERROR := FALSE;
   CP7.SP3 := FALSE;
   CP7.SP4 := FALSE;
   CP7.FC2_STATUS := W#16#0;
   CP7.FC2_DPSTATUS := B#16#0;
   CP7.FC1_STATUS := W#16#0;
   CP7.SP5 := W#16#0;
   CP7.SFC20_1_RET_VAL := 0;
   CP7.SFC20_2_RET_VAL := 0;
   CP7.SFC20_3_RET_VAL := 0;
   CP7.SFC20_4_RET_VAL := 0;
   CP7.SFC20_5_RET_VAL := 0;
   CP7.SFC20_6_RET_VAL := 0;
   CP7.SFC20_7_RET_VAL := 0;
   CP7.SFC20_8_RET_VAL := 0;
   CP7.SFC20_9_RET_VAL := 0;
   CP7.SFC20_10_RET_VAL := 0;
   CP7.SP[0] := W#16#0;
   CP7.SP[1] := W#16#0;
   CP7.SP[2] := W#16#0;
   CP7.SP[3] := W#16#0;
   CP7.SP[4] := W#16#0;
   CP7.SP[5] := W#16#0;
   CP7.SP[6] := W#16#0;
   CP7.SP[7] := W#16#0;
   CP7.SP[8] := W#16#0;
   CP7.SP[9] := W#16#0;
   CP8.FC2_NDR := FALSE;
   CP8.FC2_ERROR := FALSE;
   CP8.SP1 := FALSE;
   CP8.SP2 := FALSE;
   CP8.FC1_NDR := FALSE;
   CP8.FC1_ERROR := FALSE;
   CP8.SP3 := FALSE;
   CP8.SP4 := FALSE;
   CP8.FC2_STATUS := W#16#0;
   CP8.FC2_DPSTATUS := B#16#0;
   CP8.FC1_STATUS := W#16#0;
   CP8.SP5 := W#16#0;
   CP8.SFC20_1_RET_VAL := 0;
   CP8.SFC20_2_RET_VAL := 0;
   CP8.SFC20_3_RET_VAL := 0;
   CP8.SFC20_4_RET_VAL := 0;
   CP8.SFC20_5_RET_VAL := 0;
   CP8.SFC20_6_RET_VAL := 0;
   CP8.SFC20_7_RET_VAL := 0;
   CP8.SFC20_8_RET_VAL := 0;
   CP8.SFC20_9_RET_VAL := 0;
   CP8.SFC20_10_RET_VAL := 0;
   CP8.SP[0] := W#16#0;
   CP8.SP[1] := W#16#0;
   CP8.SP[2] := W#16#0;
   CP8.SP[3] := W#16#0;
   CP8.SP[4] := W#16#0;
   CP8.SP[5] := W#16#0;
   CP8.SP[6] := W#16#0;
   CP8.SP[7] := W#16#0;
   CP8.SP[8] := W#16#0;
   CP8.SP[9] := W#16#0;
   RTN_VALUE_WORD[0] := W#16#0;
   RTN_VALUE_WORD[1] := W#16#0;
   RTN_VALUE_WORD[2] := W#16#0;
   RTN_VALUE_WORD[3] := W#16#0;
   RTN_VALUE_WORD[4] := W#16#0;
   RTN_VALUE_WORD[5] := W#16#0;
   RTN_VALUE_WORD[6] := W#16#0;
   RTN_VALUE_WORD[7] := W#16#0;
   RTN_VALUE_WORD[8] := W#16#0;
   RTN_VALUE_WORD[9] := W#16#0;
   RTN_VALUE_WORD[10] := W#16#0;
   RTN_VALUE_WORD[11] := W#16#0;
   RTN_VALUE_WORD[12] := W#16#0;
   RTN_VALUE_WORD[13] := W#16#0;
   RTN_VALUE_WORD[14] := W#16#0;
   RTN_VALUE_WORD[15] := W#16#0;
   RTN_VALUE_WORD[16] := W#16#0;
   RTN_VALUE_WORD[17] := W#16#0;
   RTN_VALUE_WORD[18] := W#16#0;
   RTN_VALUE_WORD[19] := W#16#0;
   RTN_VALUE_WORD[20] := W#16#0;
   RTN_VALUE_WORD[21] := W#16#0;
   RTN_VALUE_WORD[22] := W#16#0;
   RTN_VALUE_WORD[23] := W#16#0;
   RTN_VALUE_WORD[24] := W#16#0;
   RTN_VALUE_WORD[25] := W#16#0;
   RTN_VALUE_WORD[26] := W#16#0;
   RTN_VALUE_WORD[27] := W#16#0;
   RTN_VALUE_WORD[28] := W#16#0;
   RTN_VALUE_WORD[29] := W#16#0;
   RTN_VALUE_WORD[30] := W#16#0;
   RTN_VALUE_WORD[31] := W#16#0;
   RTN_VALUE_WORD[32] := W#16#0;
   RTN_VALUE_WORD[33] := W#16#0;
   RTN_VALUE_WORD[34] := W#16#0;
   RTN_VALUE_WORD[35] := W#16#0;
   RTN_VALUE_WORD[36] := W#16#0;
   RTN_VALUE_WORD[37] := W#16#0;
   RTN_VALUE_WORD[38] := W#16#0;
   RTN_VALUE_WORD[39] := W#16#0;
   RTN_VALUE_WORD[40] := W#16#0;
   RTN_VALUE_WORD[41] := W#16#0;
   RTN_VALUE_WORD[42] := W#16#0;
   RTN_VALUE_WORD[43] := W#16#0;
   RTN_VALUE_WORD[44] := W#16#0;
   RTN_VALUE_WORD[45] := W#16#0;
   RTN_VALUE_WORD[46] := W#16#0;
   RTN_VALUE_WORD[47] := W#16#0;
   RTN_VALUE_WORD[48] := W#16#0;
   RTN_VALUE_WORD[49] := W#16#0;
   AG1.FC6_NDR := FALSE;
   AG1.FC6_ERROR := FALSE;
   AG1.SP1 := FALSE;
   AG1.SP2 := FALSE;
   AG1.FC5_NDR := FALSE;
   AG1.FC5_ERROR := FALSE;
   AG1.SP3 := FALSE;
   AG1.SP4 := FALSE;
   AG1.FC6_STATUS := W#16#0;
   AG1.FC6_DPSTATUS := B#16#0;
   AG1.FC5_STATUS := W#16#0;
   AG1.SP5 := W#16#0;
   AG1.SFC20_1_RET_VAL := 0;
   AG1.SFC20_2_RET_VAL := 0;
   AG1.SFC20_3_RET_VAL := 0;
   AG1.SFC20_4_RET_VAL := 0;
   AG1.SFC20_5_RET_VAL := 0;
   AG1.SFC20_6_RET_VAL := 0;
   AG1.SFC20_7_RET_VAL := 0;
   AG1.SFC20_8_RET_VAL := 0;
   AG1.SFC20_9_RET_VAL := 0;
   AG1.SFC20_10_RET_VAL := 0;
   AG1.SP[0] := W#16#0;
   AG1.SP[1] := W#16#0;
   AG1.SP[2] := W#16#0;
   AG1.SP[3] := W#16#0;
   AG1.SP[4] := W#16#0;
   AG1.SP[5] := W#16#0;
   AG1.SP[6] := W#16#0;
   AG1.SP[7] := W#16#0;
   AG1.SP[8] := W#16#0;
   AG1.SP[9] := W#16#0;
   AG2.FC6_NDR := FALSE;
   AG2.FC6_ERROR := FALSE;
   AG2.SP1 := FALSE;
   AG2.SP2 := FALSE;
   AG2.FC5_NDR := FALSE;
   AG2.FC5_ERROR := FALSE;
   AG2.SP3 := FALSE;
   AG2.SP4 := FALSE;
   AG2.FC6_STATUS := W#16#0;
   AG2.FC6_DPSTATUS := B#16#0;
   AG2.FC5_STATUS := W#16#0;
   AG2.SP5 := W#16#0;
   AG2.SFC20_1_RET_VAL := 0;
   AG2.SFC20_2_RET_VAL := 0;
   AG2.SFC20_3_RET_VAL := 0;
   AG2.SFC20_4_RET_VAL := 0;
   AG2.SFC20_5_RET_VAL := 0;
   AG2.SFC20_6_RET_VAL := 0;
   AG2.SFC20_7_RET_VAL := 0;
   AG2.SFC20_8_RET_VAL := 0;
   AG2.SFC20_9_RET_VAL := 0;
   AG2.SFC20_10_RET_VAL := 0;
   AG2.SP[0] := W#16#0;
   AG2.SP[1] := W#16#0;
   AG2.SP[2] := W#16#0;
   AG2.SP[3] := W#16#0;
   AG2.SP[4] := W#16#0;
   AG2.SP[5] := W#16#0;
   AG2.SP[6] := W#16#0;
   AG2.SP[7] := W#16#0;
   AG2.SP[8] := W#16#0;
   AG2.SP[9] := W#16#0;
   AG3.FC6_NDR := FALSE;
   AG3.FC6_ERROR := FALSE;
   AG3.SP1 := FALSE;
   AG3.SP2 := FALSE;
   AG3.FC5_NDR := FALSE;
   AG3.FC5_ERROR := FALSE;
   AG3.SP3 := FALSE;
   AG3.SP4 := FALSE;
   AG3.FC6_STATUS := W#16#0;
   AG3.FC6_DPSTATUS := B#16#0;
   AG3.FC5_STATUS := W#16#0;
   AG3.SP5 := W#16#0;
   AG3.SFC20_1_RET_VAL := 0;
   AG3.SFC20_2_RET_VAL := 0;
   AG3.SFC20_3_RET_VAL := 0;
   AG3.SFC20_4_RET_VAL := 0;
   AG3.SFC20_5_RET_VAL := 0;
   AG3.SFC20_6_RET_VAL := 0;
   AG3.SFC20_7_RET_VAL := 0;
   AG3.SFC20_8_RET_VAL := 0;
   AG3.SFC20_9_RET_VAL := 0;
   AG3.SFC20_10_RET_VAL := 0;
   AG3.SP[0] := W#16#0;
   AG3.SP[1] := W#16#0;
   AG3.SP[2] := W#16#0;
   AG3.SP[3] := W#16#0;
   AG3.SP[4] := W#16#0;
   AG3.SP[5] := W#16#0;
   AG3.SP[6] := W#16#0;
   AG3.SP[7] := W#16#0;
   AG3.SP[8] := W#16#0;
   AG3.SP[9] := W#16#0;
   AG4.FC6_NDR := FALSE;
   AG4.FC6_ERROR := FALSE;
   AG4.SP1 := FALSE;
   AG4.SP2 := FALSE;
   AG4.FC5_NDR := FALSE;
   AG4.FC5_ERROR := FALSE;
   AG4.SP3 := FALSE;
   AG4.SP4 := FALSE;
   AG4.FC6_STATUS := W#16#0;
   AG4.FC6_DPSTATUS := B#16#0;
   AG4.FC5_STATUS := W#16#0;
   AG4.SP5 := W#16#0;
   AG4.SFC20_1_RET_VAL := 0;
   AG4.SFC20_2_RET_VAL := 0;
   AG4.SFC20_3_RET_VAL := 0;
   AG4.SFC20_4_RET_VAL := 0;
   AG4.SFC20_5_RET_VAL := 0;
   AG4.SFC20_6_RET_VAL := 0;
   AG4.SFC20_7_RET_VAL := 0;
   AG4.SFC20_8_RET_VAL := 0;
   AG4.SFC20_9_RET_VAL := 0;
   AG4.SFC20_10_RET_VAL := 0;
   AG4.SP[0] := W#16#0;
   AG4.SP[1] := W#16#0;
   AG4.SP[2] := W#16#0;
   AG4.SP[3] := W#16#0;
   AG4.SP[4] := W#16#0;
   AG4.SP[5] := W#16#0;
   AG4.SP[6] := W#16#0;
   AG4.SP[7] := W#16#0;
   AG4.SP[8] := W#16#0;
   AG4.SP[9] := W#16#0;
   AG5.FC6_NDR := FALSE;
   AG5.FC6_ERROR := FALSE;
   AG5.SP1 := FALSE;
   AG5.SP2 := FALSE;
   AG5.FC5_NDR := FALSE;
   AG5.FC5_ERROR := FALSE;
   AG5.SP3 := FALSE;
   AG5.SP4 := FALSE;
   AG5.FC6_STATUS := W#16#0;
   AG5.FC6_DPSTATUS := B#16#0;
   AG5.FC5_STATUS := W#16#0;
   AG5.SP5 := W#16#0;
   AG5.SFC20_1_RET_VAL := 0;
   AG5.SFC20_2_RET_VAL := 0;
   AG5.SFC20_3_RET_VAL := 0;
   AG5.SFC20_4_RET_VAL := 0;
   AG5.SFC20_5_RET_VAL := 0;
   AG5.SFC20_6_RET_VAL := 0;
   AG5.SFC20_7_RET_VAL := 0;
   AG5.SFC20_8_RET_VAL := 0;
   AG5.SFC20_9_RET_VAL := 0;
   AG5.SFC20_10_RET_VAL := 0;
   AG5.SP[0] := W#16#0;
   AG5.SP[1] := W#16#0;
   AG5.SP[2] := W#16#0;
   AG5.SP[3] := W#16#0;
   AG5.SP[4] := W#16#0;
   AG5.SP[5] := W#16#0;
   AG5.SP[6] := W#16#0;
   AG5.SP[7] := W#16#0;
   AG5.SP[8] := W#16#0;
   AG5.SP[9] := W#16#0;
   AG6.FC6_NDR := FALSE;
   AG6.FC6_ERROR := FALSE;
   AG6.SP1 := FALSE;
   AG6.SP2 := FALSE;
   AG6.FC5_NDR := FALSE;
   AG6.FC5_ERROR := FALSE;
   AG6.SP3 := FALSE;
   AG6.SP4 := FALSE;
   AG6.FC6_STATUS := W#16#0;
   AG6.FC6_DPSTATUS := B#16#0;
   AG6.FC5_STATUS := W#16#0;
   AG6.SP5 := W#16#0;
   AG6.SFC20_1_RET_VAL := 0;
   AG6.SFC20_2_RET_VAL := 0;
   AG6.SFC20_3_RET_VAL := 0;
   AG6.SFC20_4_RET_VAL := 0;
   AG6.SFC20_5_RET_VAL := 0;
   AG6.SFC20_6_RET_VAL := 0;
   AG6.SFC20_7_RET_VAL := 0;
   AG6.SFC20_8_RET_VAL := 0;
   AG6.SFC20_9_RET_VAL := 0;
   AG6.SFC20_10_RET_VAL := 0;
   AG6.SP[0] := W#16#0;
   AG6.SP[1] := W#16#0;
   AG6.SP[2] := W#16#0;
   AG6.SP[3] := W#16#0;
   AG6.SP[4] := W#16#0;
   AG6.SP[5] := W#16#0;
   AG6.SP[6] := W#16#0;
   AG6.SP[7] := W#16#0;
   AG6.SP[8] := W#16#0;
   AG6.SP[9] := W#16#0;
   AG7.FC6_NDR := FALSE;
   AG7.FC6_ERROR := FALSE;
   AG7.SP1 := FALSE;
   AG7.SP2 := FALSE;
   AG7.FC5_NDR := FALSE;
   AG7.FC5_ERROR := FALSE;
   AG7.SP3 := FALSE;
   AG7.SP4 := FALSE;
   AG7.FC6_STATUS := W#16#0;
   AG7.FC6_DPSTATUS := B#16#0;
   AG7.FC5_STATUS := W#16#0;
   AG7.SP5 := W#16#0;
   AG7.SFC20_1_RET_VAL := 0;
   AG7.SFC20_2_RET_VAL := 0;
   AG7.SFC20_3_RET_VAL := 0;
   AG7.SFC20_4_RET_VAL := 0;
   AG7.SFC20_5_RET_VAL := 0;
   AG7.SFC20_6_RET_VAL := 0;
   AG7.SFC20_7_RET_VAL := 0;
   AG7.SFC20_8_RET_VAL := 0;
   AG7.SFC20_9_RET_VAL := 0;
   AG7.SFC20_10_RET_VAL := 0;
   AG7.SP[0] := W#16#0;
   AG7.SP[1] := W#16#0;
   AG7.SP[2] := W#16#0;
   AG7.SP[3] := W#16#0;
   AG7.SP[4] := W#16#0;
   AG7.SP[5] := W#16#0;
   AG7.SP[6] := W#16#0;
   AG7.SP[7] := W#16#0;
   AG7.SP[8] := W#16#0;
   AG7.SP[9] := W#16#0;
   SP[0] := W#16#0;
   SP[1] := W#16#0;
   SP[2] := W#16#0;
   SP[3] := W#16#0;
   SP[4] := W#16#0;
   SP[5] := W#16#0;
   SP[6] := W#16#0;
   SP[7] := W#16#0;
   SP[8] := W#16#0;
   SP[9] := W#16#0;
   SP[10] := W#16#0;
   SP[11] := W#16#0;
   SP[12] := W#16#0;
   SP[13] := W#16#0;
   SP[14] := W#16#0;
   SP[15] := W#16#0;
   SP[16] := W#16#0;
   SP[17] := W#16#0;
   SP[18] := W#16#0;
   SP[19] := W#16#0;
   SP[20] := W#16#0;
   SP[21] := W#16#0;
   SP[22] := W#16#0;
   SP[23] := W#16#0;
   SP[24] := W#16#0;
   SP[25] := W#16#0;
   SP[26] := W#16#0;
   SP[27] := W#16#0;
   SP[28] := W#16#0;
   SP[29] := W#16#0;
   SP[30] := W#16#0;
   SP[31] := W#16#0;
   SP[32] := W#16#0;
   SP[33] := W#16#0;
   SP[34] := W#16#0;
   SP[35] := W#16#0;
   SP[36] := W#16#0;
   SP[37] := W#16#0;
   SP[38] := W#16#0;
   SP[39] := W#16#0;
   SP[40] := W#16#0;
   SP[41] := W#16#0;
   SP[42] := W#16#0;
   SP[43] := W#16#0;
   SP[44] := W#16#0;
   SP[45] := W#16#0;
   SP[46] := W#16#0;
   SP[47] := W#16#0;
   SP[48] := W#16#0;
   SP[49] := W#16#0;
   SP[50] := W#16#0;
   SP[51] := W#16#0;
   SP[52] := W#16#0;
   SP[53] := W#16#0;
   SP[54] := W#16#0;
   SP[55] := W#16#0;
   SP[56] := W#16#0;
   SP[57] := W#16#0;
   SP[58] := W#16#0;
   SP[59] := W#16#0;
   SP[60] := W#16#0;
   SP[61] := W#16#0;
   SP[62] := W#16#0;
   SP[63] := W#16#0;
   SP[64] := W#16#0;
   SP[65] := W#16#0;
   SP[66] := W#16#0;
   SP[67] := W#16#0;
   SP[68] := W#16#0;
   SP[69] := W#16#0;
   SP[70] := W#16#0;
   SP[71] := W#16#0;
   SP[72] := W#16#0;
   SP[73] := W#16#0;
   SP[74] := W#16#0;
   CTYPE_RET_VAL[0] := 0;
   CTYPE_RET_VAL[1] := 0;
   CTYPE_RET_VAL[2] := 0;
   CTYPE_RET_VAL[3] := 0;
   CTYPE_RET_VAL[4] := 0;
   CTYPE_RET_VAL[5] := 0;
   CTYPE_RET_VAL[6] := 0;
   CTYPE_RET_VAL[7] := 0;
   CTYPE_RET_VAL[8] := 0;
   CTYPE_RET_VAL[9] := 0;
   CTYPE_RET_VAL[10] := 0;
   CTYPE_RET_VAL[11] := 0;
   CTYPE_RET_VAL[12] := 0;
   CTYPE_RET_VAL[13] := 0;
   CTYPE_RET_VAL[14] := 0;
   CTYPE_RET_VAL[15] := 0;
   CTYPE_RET_VAL[16] := 0;
   CTYPE_RET_VAL[17] := 0;
   CTYPE_RET_VAL[18] := 0;
   CTYPE_RET_VAL[19] := 0;
   CTYPE_RET_VAL[20] := 0;
   CTYPE_RET_VAL[21] := 0;
   CTYPE_RET_VAL[22] := 0;
   CTYPE_RET_VAL[23] := 0;
   CTYPE_RET_VAL[24] := 0;
   CTYPE_RET_VAL[25] := 0;
   CTYPE_RET_VAL[26] := 0;
   CTYPE_RET_VAL[27] := 0;
   CTYPE_RET_VAL[28] := 0;
   CTYPE_RET_VAL[29] := 0;
   CTYPE_RET_VAL[30] := 0;
   CTYPE_RET_VAL[31] := 0;
   CTYPE_RET_VAL[32] := 0;
   CTYPE_RET_VAL[33] := 0;
   CTYPE_RET_VAL[34] := 0;
   CTYPE_RET_VAL[35] := 0;
   CTYPE_RET_VAL[36] := 0;
   CTYPE_RET_VAL[37] := 0;
   CTYPE_RET_VAL[38] := 0;
   CTYPE_RET_VAL[39] := 0;
   CTYPE_RET_VAL[40] := 0;
   CTYPE_RET_VAL[41] := 0;
   CTYPE_RET_VAL[42] := 0;
   CTYPE_RET_VAL[43] := 0;
   CTYPE_RET_VAL[44] := 0;
   CTYPE_RET_VAL[45] := 0;
   CTYPE_RET_VAL[46] := 0;
   CTYPE_RET_VAL[47] := 0;
   CTYPE_RET_VAL[48] := 0;
   CTYPE_RET_VAL[49] := 0;
   CTYPE_RET_VAL[50] := 0;
   CTYPE_RET_VAL[51] := 0;
   CTYPE_RET_VAL[52] := 0;
   CTYPE_RET_VAL[53] := 0;
   CTYPE_RET_VAL[54] := 0;
   CTYPE_RET_VAL[55] := 0;
   CTYPE_RET_VAL[56] := 0;
   CTYPE_RET_VAL[57] := 0;
   CTYPE_RET_VAL[58] := 0;
   CTYPE_RET_VAL[59] := 0;
   CTYPE_RET_VAL[60] := 0;
   CTYPE_RET_VAL[61] := 0;
   CTYPE_RET_VAL[62] := 0;
   CTYPE_RET_VAL[63] := 0;
   CTYPE_RET_VAL[64] := 0;
   CTYPE_RET_VAL[65] := 0;
   CTYPE_RET_VAL[66] := 0;
   CTYPE_RET_VAL[67] := 0;
   CTYPE_RET_VAL[68] := 0;
   CTYPE_RET_VAL[69] := 0;
   CTYPE_RET_VAL[70] := 0;
   CTYPE_RET_VAL[71] := 0;
   CTYPE_RET_VAL[72] := 0;
   CTYPE_RET_VAL[73] := 0;
   CTYPE_RET_VAL[74] := 0;
   CTYPE_RET_VAL[75] := 0;
   CTYPE_RET_VAL[76] := 0;
   CTYPE_RET_VAL[77] := 0;
   CTYPE_RET_VAL[78] := 0;
   CTYPE_RET_VAL[79] := 0;
   CTYPE_RET_VAL[80] := 0;
   CTYPE_RET_VAL[81] := 0;
   CTYPE_RET_VAL[82] := 0;
   CTYPE_RET_VAL[83] := 0;
   CTYPE_RET_VAL[84] := 0;
   CTYPE_RET_VAL[85] := 0;
   CTYPE_RET_VAL[86] := 0;
   CTYPE_RET_VAL[87] := 0;
   CTYPE_RET_VAL[88] := 0;
   CTYPE_RET_VAL[89] := 0;
   CTYPE_RET_VAL[90] := 0;
   CTYPE_RET_VAL[91] := 0;
   CTYPE_RET_VAL[92] := 0;
   CTYPE_RET_VAL[93] := 0;
   CTYPE_RET_VAL[94] := 0;
   CTYPE_RET_VAL[95] := 0;
   CTYPE_RET_VAL[96] := 0;
   CTYPE_RET_VAL[97] := 0;
   CTYPE_RET_VAL[98] := 0;
   CTYPE_RET_VAL[99] := 0;
   MES_RET_VAL1[0] := 0;
   MES_RET_VAL1[1] := 0;
   MES_RET_VAL1[2] := 0;
   MES_RET_VAL1[3] := 0;
   MES_RET_VAL1[4] := 0;
   MES_RET_VAL1[5] := 0;
   MES_RET_VAL1[6] := 0;
   MES_RET_VAL1[7] := 0;
   MES_RET_VAL1[8] := 0;
   MES_RET_VAL1[9] := 0;
   MES_RET_VAL1[10] := 0;
   MES_RET_VAL1[11] := 0;
   MES_RET_VAL1[12] := 0;
   MES_RET_VAL1[13] := 0;
   MES_RET_VAL1[14] := 0;
   MES_RET_VAL1[15] := 0;
   MES_RET_VAL1[16] := 0;
   MES_RET_VAL1[17] := 0;
   MES_RET_VAL1[18] := 0;
   MES_RET_VAL1[19] := 0;
   MES_RET_VAL1[20] := 0;
   MES_RET_VAL1[21] := 0;
   MES_RET_VAL1[22] := 0;
   MES_RET_VAL1[23] := 0;
   MES_RET_VAL1[24] := 0;
   MES_RET_VAL1[25] := 0;
   MES_RET_VAL1[26] := 0;
   MES_RET_VAL1[27] := 0;
   MES_RET_VAL1[28] := 0;
   MES_RET_VAL1[29] := 0;
   MES_RET_VAL1[30] := 0;
   MES_RET_VAL1[31] := 0;
   MES_RET_VAL1[32] := 0;
   MES_RET_VAL1[33] := 0;
   MES_RET_VAL1[34] := 0;
   MES_RET_VAL1[35] := 0;
   MES_RET_VAL1[36] := 0;
   MES_RET_VAL1[37] := 0;
   MES_RET_VAL1[38] := 0;
   MES_RET_VAL1[39] := 0;
   MES_RET_VAL1[40] := 0;
   MES_RET_VAL1[41] := 0;
   MES_RET_VAL1[42] := 0;
   MES_RET_VAL1[43] := 0;
   MES_RET_VAL1[44] := 0;
   MES_RET_VAL1[45] := 0;
   MES_RET_VAL1[46] := 0;
   MES_RET_VAL1[47] := 0;
   MES_RET_VAL1[48] := 0;
   MES_RET_VAL1[49] := 0;
   MES_RET_VAL1[50] := 0;
   MES_RET_VAL1[51] := 0;
   MES_RET_VAL1[52] := 0;
   MES_RET_VAL1[53] := 0;
   MES_RET_VAL1[54] := 0;
   MES_RET_VAL1[55] := 0;
   MES_RET_VAL1[56] := 0;
   MES_RET_VAL1[57] := 0;
   MES_RET_VAL1[58] := 0;
   MES_RET_VAL1[59] := 0;
   MES_RET_VAL1[60] := 0;
   MES_RET_VAL1[61] := 0;
   MES_RET_VAL1[62] := 0;
   MES_RET_VAL1[63] := 0;
   MES_RET_VAL1[64] := 0;
   MES_RET_VAL1[65] := 0;
   MES_RET_VAL1[66] := 0;
   MES_RET_VAL1[67] := 0;
   MES_RET_VAL1[68] := 0;
   MES_RET_VAL1[69] := 0;
   MES_RET_VAL1[70] := 0;
   MES_RET_VAL1[71] := 0;
   MES_RET_VAL1[72] := 0;
   MES_RET_VAL1[73] := 0;
   MES_RET_VAL1[74] := 0;
   MES_RET_VAL1[75] := 0;
   MES_RET_VAL1[76] := 0;
   MES_RET_VAL1[77] := 0;
   MES_RET_VAL1[78] := 0;
   MES_RET_VAL1[79] := 0;
   MES_RET_VAL1[80] := 0;
   MES_RET_VAL1[81] := 0;
   MES_RET_VAL1[82] := 0;
   MES_RET_VAL1[83] := 0;
   MES_RET_VAL1[84] := 0;
   MES_RET_VAL1[85] := 0;
   MES_RET_VAL1[86] := 0;
   MES_RET_VAL1[87] := 0;
   MES_RET_VAL1[88] := 0;
   MES_RET_VAL1[89] := 0;
   MES_RET_VAL1[90] := 0;
   MES_RET_VAL1[91] := 0;
   MES_RET_VAL1[92] := 0;
   MES_RET_VAL1[93] := 0;
   MES_RET_VAL1[94] := 0;
   MES_RET_VAL1[95] := 0;
   MES_RET_VAL1[96] := 0;
   MES_RET_VAL1[97] := 0;
   MES_RET_VAL1[98] := 0;
   MES_RET_VAL1[99] := 0;
   MES_RET_VAL1[100] := 0;
   MES_RET_VAL1[101] := 0;
   MES_RET_VAL1[102] := 0;
   MES_RET_VAL1[103] := 0;
   MES_RET_VAL1[104] := 0;
   MES_RET_VAL1[105] := 0;
   MES_RET_VAL1[106] := 0;
   MES_RET_VAL1[107] := 0;
   MES_RET_VAL1[108] := 0;
   MES_RET_VAL1[109] := 0;
   MES_RET_VAL1[110] := 0;
   MES_RET_VAL1[111] := 0;
   MES_RET_VAL1[112] := 0;
   MES_RET_VAL1[113] := 0;
   MES_RET_VAL1[114] := 0;
   MES_RET_VAL1[115] := 0;
   MES_RET_VAL1[116] := 0;
   MES_RET_VAL1[117] := 0;
   MES_RET_VAL1[118] := 0;
   MES_RET_VAL1[119] := 0;
   MES_RET_VAL1[120] := 0;
   MES_RET_VAL1[121] := 0;
   MES_RET_VAL1[122] := 0;
   MES_RET_VAL1[123] := 0;
   MES_RET_VAL1[124] := 0;
   MES_RET_VAL1[125] := 0;
   MES_RET_VAL1[126] := 0;
   MES_RET_VAL1[127] := 0;
   MES_RET_VAL1[128] := 0;
   MES_RET_VAL1[129] := 0;
   MES_RET_VAL1[130] := 0;
   MES_RET_VAL1[131] := 0;
   MES_RET_VAL1[132] := 0;
   MES_RET_VAL1[133] := 0;
   MES_RET_VAL1[134] := 0;
   MES_RET_VAL1[135] := 0;
   MES_RET_VAL1[136] := 0;
   MES_RET_VAL1[137] := 0;
   MES_RET_VAL1[138] := 0;
   MES_RET_VAL1[139] := 0;
   MES_RET_VAL1[140] := 0;
   MES_RET_VAL1[141] := 0;
   MES_RET_VAL1[142] := 0;
   MES_RET_VAL1[143] := 0;
   MES_RET_VAL1[144] := 0;
   MES_RET_VAL1[145] := 0;
   MES_RET_VAL1[146] := 0;
   MES_RET_VAL1[147] := 0;
   MES_RET_VAL1[148] := 0;
   MES_RET_VAL1[149] := 0;
   MES_RET_VAL1[150] := 0;
   MES_RET_VAL1[151] := 0;
   MES_RET_VAL1[152] := 0;
   MES_RET_VAL1[153] := 0;
   MES_RET_VAL1[154] := 0;
   MES_RET_VAL1[155] := 0;
   MES_RET_VAL1[156] := 0;
   MES_RET_VAL1[157] := 0;
   MES_RET_VAL1[158] := 0;
   MES_RET_VAL1[159] := 0;
   MES_RET_VAL1[160] := 0;
   MES_RET_VAL1[161] := 0;
   MES_RET_VAL1[162] := 0;
   MES_RET_VAL1[163] := 0;
   MES_RET_VAL1[164] := 0;
   MES_RET_VAL1[165] := 0;
   MES_RET_VAL1[166] := 0;
   MES_RET_VAL1[167] := 0;
   MES_RET_VAL1[168] := 0;
   MES_RET_VAL1[169] := 0;
   MES_RET_VAL1[170] := 0;
   MES_RET_VAL1[171] := 0;
   MES_RET_VAL1[172] := 0;
   MES_RET_VAL1[173] := 0;
   MES_RET_VAL1[174] := 0;
   MES_RET_VAL1[175] := 0;
   MES_RET_VAL1[176] := 0;
   MES_RET_VAL1[177] := 0;
   MES_RET_VAL1[178] := 0;
   MES_RET_VAL1[179] := 0;
   MES_RET_VAL1[180] := 0;
   MES_RET_VAL1[181] := 0;
   MES_RET_VAL1[182] := 0;
   MES_RET_VAL1[183] := 0;
   MES_RET_VAL1[184] := 0;
   MES_RET_VAL1[185] := 0;
   MES_RET_VAL1[186] := 0;
   MES_RET_VAL1[187] := 0;
   MES_RET_VAL1[188] := 0;
   MES_RET_VAL1[189] := 0;
   MES_RET_VAL1[190] := 0;
   MES_RET_VAL1[191] := 0;
   MES_RET_VAL1[192] := 0;
   MES_RET_VAL1[193] := 0;
   MES_RET_VAL1[194] := 0;
   MES_RET_VAL1[195] := 0;
   MES_RET_VAL1[196] := 0;
   MES_RET_VAL1[197] := 0;
   MES_RET_VAL1[198] := 0;
   MES_RET_VAL1[199] := 0;
END_DATA_BLOCK

DATA_BLOCK DB 60
TITLE =
VERSION : 0.1


